LIN {X 0,Y 740.172,Z 409.434,A -85,B 0,C 180,E1 27946.505,E2 27946.505} C_VEL
LIN {X 0,Y 736.938,Z 402.446,A -85,B 0,C 180,E1 27945.781,E2 27945.781} C_VEL
LIN {X 0,Y 735.986,Z 399.553,A -85,B 0,C 180,E1 27945.49,E2 27945.49} C_VEL
LIN {X 0,Y 735.996,Z 399.549,A -85,B 0,C 180,E1 27943.152,E2 27943.152} C_VEL
LIN {X 0,Y 736.087,Z 399.542,A -85,B 0,C 180,E1 27940.285,E2 27940.285} C_VEL
LIN {X 0,Y 736.005,Z 399.54,A -85,B 0,C 180,E1 27937.589,E2 27937.589} C_VEL
LIN {X 0,Y 736,Z 399.544,A -85,B 0,C 180,E1 27935.266,E2 27935.266} C_VEL
LIN {X 0,Y 736.007,Z 399.541,A -85,B 0,C 180,E1 27933.009,E2 27933.009} C_VEL
LIN {X 0,Y 736.096,Z 399.538,A -85,B 0,C 180,E1 27930.24,E2 27930.24} C_VEL
LIN {X 0,Y 736.029,Z 399.541,A -85,B 0,C 180,E1 27927.421,E2 27927.421} C_VEL
LIN {X 0,Y 736.015,Z 399.535,A -85,B 0,C 180,E1 27924.993,E2 27924.993} C_VEL
LIN {X 0,Y 736.039,Z 399.543,A -85,B 0,C 180,E1 27922.518,E2 27922.518} C_VEL
LIN {X 0,Y 736.074,Z 399.535,A -85,B 0,C 180,E1 27919.485,E2 27919.485} C_VEL
LIN {X 0,Y 736.029,Z 399.54,A -85,B 0,C 180,E1 27916.82,E2 27916.82} C_VEL
LIN {X 0,Y 736.059,Z 399.536,A -85,B 0,C 180,E1 27914.234,E2 27914.234} C_VEL
LIN {X 0,Y 736.066,Z 399.535,A -85,B 0,C 180,E1 27911.122,E2 27911.122} C_VEL
LIN {X 0,Y 736.042,Z 399.533,A -85,B 0,C 180,E1 27908.437,E2 27908.437} C_VEL
LIN {X 0,Y 736.098,Z 399.541,A -85,B 0,C 180,E1 27905.691,E2 27905.691} C_VEL
LIN {X 0,Y 736.059,Z 399.529,A -85,B 0,C 180,E1 27902.725,E2 27902.725} C_VEL
LIN {X 0,Y 736.072,Z 399.542,A -85,B 0,C 180,E1 27899.922,E2 27899.922} C_VEL
LIN {X 0,Y 736.095,Z 399.525,A -85,B 0,C 180,E1 27896.885,E2 27896.885} C_VEL
LIN {X 0,Y 736.064,Z 399.54,A -85,B 0,C 180,E1 27893.996,E2 27893.996} C_VEL
LIN {X 0,Y 736.084,Z 399.532,A -85,B 0,C 180,E1 27891.17,E2 27891.17} C_VEL
LIN {X 0,Y 736.082,Z 399.538,A -85,B 0,C 180,E1 27889.085,E2 27889.085} C_VEL
LIN {X 0,Y 735.104,Z 399.658,A -85,B 0,C 180,E1 27888.486,E2 27888.486} C_VEL
LIN {X 0,Y 728.704,Z 400.452,A -85,B 0,C 180,E1 27886.806,E2 27886.806} C_VEL
LIN {X 0,Y 728.145,Z 400.519,A -85,B 0,C 180,E1 27886.37,E2 27886.37} C_VEL
LIN {X 0,Y 728.158,Z 400.528,A -85,B 0,C 180,E1 27883.404,E2 27883.404} C_VEL
LIN {X 0,Y 728.158,Z 400.516,A -85,B 0,C 180,E1 27880.34,E2 27880.34} C_VEL
LIN {X 0,Y 728.159,Z 400.532,A -85,B 0,C 180,E1 27877.303,E2 27877.303} C_VEL
LIN {X 0,Y 728.149,Z 400.514,A -85,B 0,C 180,E1 27874.265,E2 27874.265} C_VEL
LIN {X 0,Y 728.155,Z 400.529,A -85,B 0,C 180,E1 27871.174,E2 27871.174} C_VEL
LIN {X 0,Y 728.136,Z 400.524,A -85,B 0,C 180,E1 27868.214,E2 27868.214} C_VEL
LIN {X 0,Y 728.153,Z 400.524,A -85,B 0,C 180,E1 27865.202,E2 27865.202} C_VEL
LIN {X 0,Y 728.116,Z 400.521,A -85,B 0,C 180,E1 27862.331,E2 27862.331} C_VEL
LIN {X 0,Y 728.157,Z 400.526,A -85,B 0,C 180,E1 27859.495,E2 27859.495} C_VEL
LIN {X 0,Y 728.12,Z 400.535,A -85,B 0,C 180,E1 27856.528,E2 27856.528} C_VEL
LIN {X 0,Y 728.127,Z 400.666,A -85,B 0,C 180,E1 27854.303,E2 27854.303} C_VEL
LIN {X 0,Y 729.384,Z 403.968,A -85,B 0,C 180,E1 27853.969,E2 27853.969} C_VEL
LIN {X 0,Y 733.459,Z 413.169,A -85,B 0,C 180,E1 27853.013,E2 27853.013} C_VEL
LIN {X 0,Y 733.539,Z 418.371,A -85,B 0,C 180,E1 27852.673,E2 27852.673} C_VEL
LIN {X 0,Y 735.86,Z 427.418,A -85,B 0,C 180,E1 27852.39,E2 27852.39} C_VEL
LIN {X 0,Y 734.932,Z 640.42,A -85,B 0,C 180,E1 27849.748,E2 27849.748} C_VEL
LIN {X 0,Y 734.045,Z 865.401,A -85,B 0,C 180,E1 27847.051,E2 27847.051} C_VEL
LIN {X 0,Y 733.84,Z 901.954,A -85,B 0,C 180,E1 27846.581,E2 27846.581} C_VEL
LIN {X 0,Y 733.507,Z 929.139,A -85,B 0,C 180,E1 27846.067,E2 27846.067} C_VEL
LIN {X 0,Y 733.146,Z 955.092,A -85,B 0,C 180,E1 27845.422,E2 27845.422} C_VEL
LIN {X 0,Y 732.693,Z 983.223,A -85,B 0,C 180,E1 27844.544,E2 27844.544} C_VEL
LIN {X 0,Y 732.219,Z 1006.493,A -85,B 0,C 180,E1 27843.671,E2 27843.671} C_VEL
LIN {X 0,Y 731.801,Z 1027.689,A -85,B 0,C 180,E1 27842.757,E2 27842.757} C_VEL
LIN {X 0,Y 731.382,Z 1048.987,A -85,B 0,C 180,E1 27841.718,E2 27841.718} C_VEL
LIN {X 0,Y 730.847,Z 1074.292,A -85,B 0,C 180,E1 27840.312,E2 27840.312} C_VEL
LIN {X 0,Y 730.375,Z 1094.539,A -85,B 0,C 180,E1 27839.034,E2 27839.034} C_VEL
LIN {X 0,Y 730.006,Z 1112.829,A -85,B 0,C 180,E1 27837.757,E2 27837.757} C_VEL
LIN {X 0,Y 729.606,Z 1134.181,A -85,B 0,C 180,E1 27836.1,E2 27836.1} C_VEL
LIN {X 0,Y 729.201,Z 1151.944,A -85,B 0,C 180,E1 27834.551,E2 27834.551} C_VEL
LIN {X 0,Y 728.96,Z 1167.07,A -85,B 0,C 180,E1 27833.099,E2 27833.099} C_VEL
LIN {X 0,Y 728.696,Z 1184.595,A -85,B 0,C 180,E1 27831.24,E2 27831.24} C_VEL
LIN {X 0,Y 728.444,Z 1199.796,A -85,B 0,C 180,E1 27829.402,E2 27829.402} C_VEL
LIN {X 0,Y 728.27,Z 1211.506,A -85,B 0,C 180,E1 27827.83,E2 27827.83} C_VEL
LIN {X 0,Y 728.154,Z 1221.964,A -85,B 0,C 180,E1 27826.269,E2 27826.269} C_VEL
LIN {X 0,Y 728.097,Z 1232.189,A -85,B 0,C 180,E1 27824.557,E2 27824.557} C_VEL
LIN {X 0,Y 728.012,Z 1243.15,A -85,B 0,C 180,E1 27822.438,E2 27822.438} C_VEL
LIN {X 0,Y 727.956,Z 1251.705,A -85,B 0,C 180,E1 27820.431,E2 27820.431} C_VEL
LIN {X 0,Y 727.918,Z 1257.897,A -85,B 0,C 180,E1 27818.692,E2 27818.692} C_VEL
LIN {X 0,Y 727.914,Z 1263.45,A -85,B 0,C 180,E1 27816.786,E2 27816.786} C_VEL
LIN {X 0,Y 727.906,Z 1267.979,A -85,B 0,C 180,E1 27814.651,E2 27814.651} C_VEL
LIN {X 0,Y 727.907,Z 1270.635,A -85,B 0,C 180,E1 27812.6,E2 27812.6} C_VEL
LIN {X 0,Y 727.87,Z 1271.746,A -85,B 0,C 180,E1 27810.868,E2 27810.868} C_VEL
LIN {X 0,Y 727.863,Z 1271.818,A -85,B 0,C 180,E1 27809.294,E2 27809.294} C_VEL
LIN {X 0,Y 727.903,Z 1270.919,A -85,B 0,C 180,E1 27807.641,E2 27807.641} C_VEL
LIN {X 0,Y 727.919,Z 1268.753,A -85,B 0,C 180,E1 27805.749,E2 27805.749} C_VEL
LIN {X 0,Y 727.925,Z 1264.66,A -85,B 0,C 180,E1 27803.614,E2 27803.614} C_VEL
LIN {X 0,Y 727.938,Z 1258.97,A -85,B 0,C 180,E1 27801.551,E2 27801.551} C_VEL
LIN {X 0,Y 727.959,Z 1252.922,A -85,B 0,C 180,E1 27799.797,E2 27799.797} C_VEL
LIN {X 0,Y 727.968,Z 1246,A -85,B 0,C 180,E1 27798.113,E2 27798.113} C_VEL
LIN {X 0,Y 727.993,Z 1238.385,A -85,B 0,C 180,E1 27796.516,E2 27796.516} C_VEL
LIN {X 0,Y 728.083,Z 1229.937,A -85,B 0,C 180,E1 27794.959,E2 27794.959} C_VEL
LIN {X 0,Y 728.214,Z 1219.431,A -85,B 0,C 180,E1 27793.244,E2 27793.244} C_VEL
LIN {X 0,Y 728.406,Z 1204.399,A -85,B 0,C 180,E1 27791.101,E2 27791.101} C_VEL
LIN {X 0,Y 728.578,Z 1190.37,A -85,B 0,C 180,E1 27789.351,E2 27789.351} C_VEL
LIN {X 0,Y 728.782,Z 1176.161,A -85,B 0,C 180,E1 27787.752,E2 27787.752} C_VEL
LIN {X 0,Y 729.149,Z 1157.625,A -85,B 0,C 180,E1 27785.884,E2 27785.884} C_VEL
LIN {X 0,Y 729.437,Z 1139.857,A -85,B 0,C 180,E1 27784.292,E2 27784.292} C_VEL
LIN {X 0,Y 729.828,Z 1122.232,A -85,B 0,C 180,E1 27782.86,E2 27782.86} C_VEL
LIN {X 0,Y 730.303,Z 1099.259,A -85,B 0,C 180,E1 27781.192,E2 27781.192} C_VEL
LIN {X 0,Y 730.687,Z 1080.033,A -85,B 0,C 180,E1 27779.948,E2 27779.948} C_VEL
LIN {X 0,Y 731.122,Z 1060.07,A -85,B 0,C 180,E1 27778.784,E2 27778.784} C_VEL
LIN {X 0,Y 731.711,Z 1035.688,A -85,B 0,C 180,E1 27777.522,E2 27777.522} C_VEL
LIN {X 0,Y 732.155,Z 1010.998,A -85,B 0,C 180,E1 27776.425,E2 27776.425} C_VEL
LIN {X 0,Y 732.522,Z 990.893,A -85,B 0,C 180,E1 27775.642,E2 27775.642} C_VEL
LIN {X 0,Y 732.878,Z 969.752,A -85,B 0,C 180,E1 27774.927,E2 27774.927} C_VEL
LIN {X 0,Y 733.272,Z 946.183,A -85,B 0,C 180,E1 27774.25,E2 27774.25} C_VEL
LIN {X 0,Y 733.633,Z 919.552,A -85,B 0,C 180,E1 27773.644,E2 27773.644} C_VEL
LIN {X 0,Y 733.894,Z 892.765,A -85,B 0,C 180,E1 27773.194,E2 27773.194} C_VEL
LIN {X 0,Y 734.857,Z 657.43,A -85,B 0,C 180,E1 27770.369,E2 27770.369} C_VEL
LIN {X 0,Y 735.717,Z 452.431,A -85,B 0,C 180,E1 27767.834,E2 27767.834} C_VEL
LIN {X 0,Y 735.682,Z 426.075,A -85,B 0,C 180,E1 27767.49,E2 27767.49} C_VEL
LIN {X 0,Y 733.393,Z 417.703,A -85,B 0,C 180,E1 27767.209,E2 27767.209} C_VEL
LIN {X 0,Y 733.27,Z 412.662,A -85,B 0,C 180,E1 27766.847,E2 27766.847} C_VEL
LIN {X 0,Y 728.891,Z 403.155,A -85,B 0,C 180,E1 27765.845,E2 27765.845} C_VEL
LIN {X 0,Y 728.094,Z 400.538,A -85,B 0,C 180,E1 27765.571,E2 27765.571} C_VEL
LIN {X 0,Y 728.16,Z 400.529,A -85,B 0,C 180,E1 27762.715,E2 27762.715} C_VEL
LIN {X 0,Y 728.101,Z 400.53,A -85,B 0,C 180,E1 27759.862,E2 27759.862} C_VEL
LIN {X 0,Y 728.09,Z 400.531,A -85,B 0,C 180,E1 27757.339,E2 27757.339} C_VEL
LIN {X 0,Y 728.157,Z 400.524,A -85,B 0,C 180,E1 27754.53,E2 27754.53} C_VEL
LIN {X 0,Y 728.104,Z 400.526,A -85,B 0,C 180,E1 27751.641,E2 27751.641} C_VEL
LIN {X 0,Y 728.085,Z 400.526,A -85,B 0,C 180,E1 27749.088,E2 27749.088} C_VEL
LIN {X 0,Y 728.133,Z 400.532,A -85,B 0,C 180,E1 27746.419,E2 27746.419} C_VEL
LIN {X 0,Y 728.103,Z 400.528,A -85,B 0,C 180,E1 27743.383,E2 27743.383} C_VEL
LIN {X 0,Y 728.081,Z 400.525,A -85,B 0,C 180,E1 27740.92,E2 27740.92} C_VEL
LIN {X 0,Y 728.097,Z 400.529,A -85,B 0,C 180,E1 27738.403,E2 27738.403} C_VEL
LIN {X 0,Y 728.145,Z 400.517,A -85,B 0,C 180,E1 27735.442,E2 27735.442} C_VEL
LIN {X 0,Y 728.081,Z 400.528,A -85,B 0,C 180,E1 27732.774,E2 27732.774} C_VEL
LIN {X 0,Y 728.078,Z 400.529,A -85,B 0,C 180,E1 27730.364,E2 27730.364} C_VEL
LIN {X 0,Y 728.14,Z 400.525,A -85,B 0,C 180,E1 27727.655,E2 27727.655} C_VEL
LIN {X 0,Y 728.096,Z 400.526,A -85,B 0,C 180,E1 27724.726,E2 27724.726} C_VEL
LIN {X 0,Y 728.073,Z 400.522,A -85,B 0,C 180,E1 27722.283,E2 27722.283} C_VEL
LIN {X 0,Y 728.082,Z 400.532,A -85,B 0,C 180,E1 27719.843,E2 27719.843} C_VEL
LIN {X 0,Y 728.159,Z 400.52,A -85,B 0,C 180,E1 27716.93,E2 27716.93} C_VEL
LIN {X 0,Y 728.077,Z 400.53,A -85,B 0,C 180,E1 27714.167,E2 27714.167} C_VEL
LIN {X 0,Y 728.069,Z 400.528,A -85,B 0,C 180,E1 27711.788,E2 27711.788} C_VEL
LIN {X 0,Y 728.09,Z 400.527,A -85,B 0,C 180,E1 27709.316,E2 27709.316} C_VEL
LIN {X 0,Y 728.11,Z 400.524,A -85,B 0,C 180,E1 27706.256,E2 27706.256} C_VEL
LIN {X 0,Y 728.068,Z 400.527,A -85,B 0,C 180,E1 27703.716,E2 27703.716} C_VEL
LIN {X 0,Y 728.065,Z 400.531,A -85,B 0,C 180,E1 27701.357,E2 27701.357} C_VEL
LIN {X 0,Y 728.097,Z 400.524,A -85,B 0,C 180,E1 27698.827,E2 27698.827} C_VEL
LIN {X 0,Y 728.088,Z 400.527,A -85,B 0,C 180,E1 27695.754,E2 27695.754} C_VEL
LIN {X 0,Y 728.061,Z 400.53,A -85,B 0,C 180,E1 27693.315,E2 27693.315} C_VEL
LIN {X 0,Y 728.059,Z 400.531,A -85,B 0,C 180,E1 27691.091,E2 27691.091} C_VEL
LIN {X 0,Y 728.063,Z 400.53,A -85,B 0,C 180,E1 27688.817,E2 27688.817} C_VEL
LIN {X 0,Y 728.149,Z 400.526,A -85,B 0,C 180,E1 27686.03,E2 27686.03} C_VEL
LIN {X 0,Y 728.07,Z 400.533,A -85,B 0,C 180,E1 27683.186,E2 27683.186} C_VEL
LIN {X 0,Y 728.055,Z 400.535,A -85,B 0,C 180,E1 27680.82,E2 27680.82} C_VEL
LIN {X 0,Y 728.054,Z 400.529,A -85,B 0,C 180,E1 27678.55,E2 27678.55} C_VEL
LIN {X 0,Y 728.081,Z 400.539,A -85,B 0,C 180,E1 27676.09,E2 27676.09} C_VEL
LIN {X 0,Y 728.109,Z 400.757,A -85,B 0,C 180,E1 27675.02,E2 27675.02} C_VEL
LIN {X 0,Y 729.543,Z 404.285,A -85,B 0,C 180,E1 27674.657,E2 27674.657} C_VEL
LIN {X 0,Y 733.638,Z 413.428,A -85,B 0,C 180,E1 27673.704,E2 27673.704} C_VEL
LIN {X 0,Y 733.606,Z 428.254,A -85,B 0,C 180,E1 27672.715,E2 27672.715} C_VEL
LIN {X 0,Y 735.808,Z 437.166,A -85,B 0,C 180,E1 27672.442,E2 27672.442} C_VEL
LIN {X 0,Y 734.994,Z 637.58,A -85,B 0,C 180,E1 27669.949,E2 27669.949} C_VEL
LIN {X 0,Y 734.094,Z 863.168,A -85,B 0,C 180,E1 27667.24,E2 27667.24} C_VEL
LIN {X 0,Y 733.848,Z 909.112,A -85,B 0,C 180,E1 27666.669,E2 27666.669} C_VEL
LIN {X 0,Y 733.533,Z 936.271,A -85,B 0,C 180,E1 27666.174,E2 27666.174} C_VEL
LIN {X 0,Y 733.191,Z 962.414,A -85,B 0,C 180,E1 27665.54,E2 27665.54} C_VEL
LIN {X 0,Y 732.806,Z 987.825,A -85,B 0,C 180,E1 27664.77,E2 27664.77} C_VEL
LIN {X 0,Y 732.285,Z 1014.336,A -85,B 0,C 180,E1 27663.804,E2 27663.804} C_VEL
LIN {X 0,Y 731.832,Z 1035.781,A -85,B 0,C 180,E1 27662.89,E2 27662.89} C_VEL
LIN {X 0,Y 731.418,Z 1056.259,A -85,B 0,C 180,E1 27661.903,E2 27661.903} C_VEL
LIN {X 0,Y 730.988,Z 1078.915,A -85,B 0,C 180,E1 27660.674,E2 27660.674} C_VEL
LIN {X 0,Y 730.433,Z 1102.632,A -85,B 0,C 180,E1 27659.206,E2 27659.206} C_VEL
LIN {X 0,Y 730.019,Z 1121.699,A -85,B 0,C 180,E1 27657.884,E2 27657.884} C_VEL
LIN {X 0,Y 729.65,Z 1141.909,A -85,B 0,C 180,E1 27656.334,E2 27656.334} C_VEL
LIN {X 0,Y 729.212,Z 1161.552,A -85,B 0,C 180,E1 27654.632,E2 27654.632} C_VEL
LIN {X 0,Y 728.956,Z 1177.569,A -85,B 0,C 180,E1 27653.094,E2 27653.094} C_VEL
LIN {X 0,Y 728.684,Z 1195.015,A -85,B 0,C 180,E1 27651.235,E2 27651.235} C_VEL
LIN {X 0,Y 728.438,Z 1210.181,A -85,B 0,C 180,E1 27649.398,E2 27649.398} C_VEL
LIN {X 0,Y 728.264,Z 1221.856,A -85,B 0,C 180,E1 27647.826,E2 27647.826} C_VEL
LIN {X 0,Y 728.149,Z 1232.802,A -85,B 0,C 180,E1 27646.183,E2 27646.183} C_VEL
LIN {X 0,Y 728.085,Z 1244.324,A -85,B 0,C 180,E1 27644.227,E2 27644.227} C_VEL
LIN {X 0,Y 727.973,Z 1254.727,A -85,B 0,C 180,E1 27642.128,E2 27642.128} C_VEL
LIN {X 0,Y 727.956,Z 1261.878,A -85,B 0,C 180,E1 27640.431,E2 27640.431} C_VEL
LIN {X 0,Y 727.915,Z 1267.801,A -85,B 0,C 180,E1 27638.768,E2 27638.768} C_VEL
LIN {X 0,Y 727.918,Z 1273.181,A -85,B 0,C 180,E1 27636.94,E2 27636.94} C_VEL
LIN {X 0,Y 727.911,Z 1277.787,A -85,B 0,C 180,E1 27634.804,E2 27634.804} C_VEL
LIN {X 0,Y 727.913,Z 1280.543,A -85,B 0,C 180,E1 27632.753,E2 27632.753} C_VEL
LIN {X 0,Y 727.874,Z 1281.715,A -85,B 0,C 180,E1 27631.021,E2 27631.021} C_VEL
LIN {X 0,Y 727.863,Z 1281.826,A -85,B 0,C 180,E1 27629.368,E2 27629.368} C_VEL
LIN {X 0,Y 727.907,Z 1280.944,A -85,B 0,C 180,E1 27627.715,E2 27627.715} C_VEL
LIN {X 0,Y 727.919,Z 1278.799,A -85,B 0,C 180,E1 27625.823,E2 27625.823} C_VEL
LIN {X 0,Y 727.925,Z 1274.73,A -85,B 0,C 180,E1 27623.689,E2 27623.689} C_VEL
LIN {X 0,Y 727.94,Z 1269.067,A -85,B 0,C 180,E1 27621.626,E2 27621.626} C_VEL
LIN {X 0,Y 727.957,Z 1263.038,A -85,B 0,C 180,E1 27619.872,E2 27619.872} C_VEL
LIN {X 0,Y 727.966,Z 1256.136,A -85,B 0,C 180,E1 27618.189,E2 27618.189} C_VEL
LIN {X 0,Y 727.992,Z 1248.874,A -85,B 0,C 180,E1 27616.657,E2 27616.657} C_VEL
LIN {X 0,Y 728.086,Z 1240.585,A -85,B 0,C 180,E1 27615.118,E2 27615.118} C_VEL
LIN {X 0,Y 728.176,Z 1230.683,A -85,B 0,C 180,E1 27613.485,E2 27613.485} C_VEL
LIN {X 0,Y 728.348,Z 1218.33,A -85,B 0,C 180,E1 27611.675,E2 27611.675} C_VEL
LIN {X 0,Y 728.544,Z 1202.255,A -85,B 0,C 180,E1 27609.617,E2 27609.617} C_VEL
LIN {X 0,Y 728.751,Z 1188.504,A -85,B 0,C 180,E1 27608.051,E2 27608.051} C_VEL
LIN {X 0,Y 729.019,Z 1173.252,A -85,B 0,C 180,E1 27606.475,E2 27606.475} C_VEL
LIN {X 0,Y 729.419,Z 1152.829,A -85,B 0,C 180,E1 27604.591,E2 27604.591} C_VEL
LIN {X 0,Y 729.707,Z 1136.033,A -85,B 0,C 180,E1 27603.203,E2 27603.203} C_VEL
LIN {X 0,Y 730.116,Z 1118.042,A -85,B 0,C 180,E1 27601.851,E2 27601.851} C_VEL
LIN {X 0,Y 730.637,Z 1095.045,A -85,B 0,C 180,E1 27600.303,E2 27600.303} C_VEL
LIN {X 0,Y 731.035,Z 1073.976,A -85,B 0,C 180,E1 27599.048,E2 27599.048} C_VEL
LIN {X 0,Y 731.459,Z 1053.715,A -85,B 0,C 180,E1 27597.967,E2 27597.967} C_VEL
LIN {X 0,Y 732.011,Z 1030.233,A -85,B 0,C 180,E1 27596.859,E2 27596.859} C_VEL
LIN {X 0,Y 732.493,Z 1004.359,A -85,B 0,C 180,E1 27595.815,E2 27595.815} C_VEL
LIN {X 0,Y 732.86,Z 982.526,A -85,B 0,C 180,E1 27595.061,E2 27595.061} C_VEL
LIN {X 0,Y 733.226,Z 959.937,A -85,B 0,C 180,E1 27594.393,E2 27594.393} C_VEL
LIN {X 0,Y 733.593,Z 933.231,A -85,B 0,C 180,E1 27593.762,E2 27593.762} C_VEL
LIN {X 0,Y 733.868,Z 905.776,A -85,B 0,C 180,E1 27593.281,E2 27593.281} C_VEL
LIN {X 0,Y 734.847,Z 670.065,A -85,B 0,C 180,E1 27590.446,E2 27590.446} C_VEL
LIN {X 0,Y 735.657,Z 471.261,A -85,B 0,C 180,E1 27587.988,E2 27587.988} C_VEL
LIN {X 0,Y 735.65,Z 435.773,A -85,B 0,C 180,E1 27587.529,E2 27587.529} C_VEL
LIN {X 0,Y 733.473,Z 427.342,A -85,B 0,C 180,E1 27587.243,E2 27587.243} C_VEL
LIN {X 0,Y 733.521,Z 413.008,A -85,B 0,C 180,E1 27586.259,E2 27586.259} C_VEL
LIN {X 0,Y 728.16,Z 401.076,A -85,B 0,C 180,E1 27585.007,E2 27585.007} C_VEL
LIN {X 0,Y 728.082,Z 400.54,A -85,B 0,C 180,E1 27584.938,E2 27584.938} C_VEL
LIN {X 0,Y 728.072,Z 400.531,A -85,B 0,C 180,E1 27581.87,E2 27581.87} C_VEL
LIN {X 0,Y 728.055,Z 400.536,A -85,B 0,C 180,E1 27579.481,E2 27579.481} C_VEL
LIN {X 0,Y 728.06,Z 400.529,A -85,B 0,C 180,E1 27577.177,E2 27577.177} C_VEL
LIN {X 0,Y 728.102,Z 400.534,A -85,B 0,C 180,E1 27574.649,E2 27574.649} C_VEL
LIN {X 0,Y 728.094,Z 400.53,A -85,B 0,C 180,E1 27571.631,E2 27571.631} C_VEL
LIN {X 0,Y 728.071,Z 400.527,A -85,B 0,C 180,E1 27569.139,E2 27569.139} C_VEL
LIN {X 0,Y 728.083,Z 400.532,A -85,B 0,C 180,E1 27566.773,E2 27566.773} C_VEL
LIN {X 0,Y 728.161,Z 400.528,A -85,B 0,C 180,E1 27563.861,E2 27563.861} C_VEL
LIN {X 0,Y 728.09,Z 400.525,A -85,B 0,C 180,E1 27561.088,E2 27561.088} C_VEL
LIN {X 0,Y 728.095,Z 400.528,A -85,B 0,C 180,E1 27558.579,E2 27558.579} C_VEL
LIN {X 0,Y 728.159,Z 400.518,A -85,B 0,C 180,E1 27555.695,E2 27555.695} C_VEL
LIN {X 0,Y 728.1,Z 400.527,A -85,B 0,C 180,E1 27552.832,E2 27552.832} C_VEL
LIN {X 0,Y 728.127,Z 400.531,A -85,B 0,C 180,E1 27550.124,E2 27550.124} C_VEL
LIN {X 0,Y 728.133,Z 400.523,A -85,B 0,C 180,E1 27547.02,E2 27547.02} C_VEL
LIN {X 0,Y 728.113,Z 400.528,A -85,B 0,C 180,E1 27544.253,E2 27544.253} C_VEL
LIN {X 0,Y 728.152,Z 400.528,A -85,B 0,C 180,E1 27541.416,E2 27541.416} C_VEL
LIN {X 0,Y 728.124,Z 400.523,A -85,B 0,C 180,E1 27538.584,E2 27538.584} C_VEL
LIN {X 0,Y 728.145,Z 400.524,A -85,B 0,C 180,E1 27535.747,E2 27535.747} C_VEL
LIN {X 0,Y 728.153,Z 400.519,A -85,B 0,C 180,E1 27532.663,E2 27532.663} C_VEL
LIN {X 0,Y 728.147,Z 400.524,A -85,B 0,C 180,E1 27529.637,E2 27529.637} C_VEL
LIN {X 0,Y 728.159,Z 400.518,A -85,B 0,C 180,E1 27526.581,E2 27526.581} C_VEL
LIN {X 0,Y 728.145,Z 400.519,A -85,B 0,C 180,E1 27526.37,E2 27526.37} C_VEL
LIN {X 0,Y 727.117,Z 400.655,A -85,B 0,C 180,E1 27525.764,E2 27525.764} C_VEL
LIN {X 0,Y 720.707,Z 401.444,A -85,B 0,C 180,E1 27524.066,E2 27524.066} C_VEL
LIN {X 0,Y 720.204,Z 401.513,A -85,B 0,C 180,E1 27523.625,E2 27523.625} C_VEL
LIN {X 0,Y 720.2,Z 401.508,A -85,B 0,C 180,E1 27520.705,E2 27520.705} C_VEL
LIN {X 0,Y 720.199,Z 401.513,A -85,B 0,C 180,E1 27517.813,E2 27517.813} C_VEL
LIN {X 0,Y 720.198,Z 401.509,A -85,B 0,C 180,E1 27514.947,E2 27514.947} C_VEL
LIN {X 0,Y 720.22,Z 401.511,A -85,B 0,C 180,E1 27512.002,E2 27512.002} C_VEL
LIN {X 0,Y 720.204,Z 401.518,A -85,B 0,C 180,E1 27508.938,E2 27508.938} C_VEL
LIN {X 0,Y 720.21,Z 401.505,A -85,B 0,C 180,E1 27505.979,E2 27505.979} C_VEL
LIN {X 0,Y 720.201,Z 401.514,A -85,B 0,C 180,E1 27502.836,E2 27502.836} C_VEL
LIN {X 0,Y 720.196,Z 401.515,A -85,B 0,C 180,E1 27499.906,E2 27499.906} C_VEL
LIN {X 0,Y 720.206,Z 401.523,A -85,B 0,C 180,E1 27496.793,E2 27496.793} C_VEL
LIN {X 0,Y 720.228,Z 401.618,A -85,B 0,C 180,E1 27494.851,E2 27494.851} C_VEL
LIN {X 0,Y 721.644,Z 405.235,A -85,B 0,C 180,E1 27494.474,E2 27494.474} C_VEL
LIN {X 0,Y 726.876,Z 417.505,A -85,B 0,C 180,E1 27493.191,E2 27493.191} C_VEL
LIN {X 0,Y 729.928,Z 429.522,A -85,B 0,C 180,E1 27492.789,E2 27492.789} C_VEL
LIN {X 0,Y 728.768,Z 641.616,A -85,B 0,C 180,E1 27490.138,E2 27490.138} C_VEL
LIN {X 0,Y 727.652,Z 866.412,A -85,B 0,C 180,E1 27487.42,E2 27487.42} C_VEL
LIN {X 0,Y 727.395,Z 902.179,A -85,B 0,C 180,E1 27486.955,E2 27486.955} C_VEL
LIN {X 0,Y 726.977,Z 929.413,A -85,B 0,C 180,E1 27486.436,E2 27486.436} C_VEL
LIN {X 0,Y 726.54,Z 955.115,A -85,B 0,C 180,E1 27485.794,E2 27485.794} C_VEL
LIN {X 0,Y 725.973,Z 983.236,A -85,B 0,C 180,E1 27484.91,E2 27484.91} C_VEL
LIN {X 0,Y 725.391,Z 1006.511,A -85,B 0,C 180,E1 27484.032,E2 27484.032} C_VEL
LIN {X 0,Y 724.843,Z 1027.705,A -85,B 0,C 180,E1 27483.112,E2 27483.112} C_VEL
LIN {X 0,Y 724.296,Z 1049.98,A -85,B 0,C 180,E1 27482.014,E2 27482.014} C_VEL
LIN {X 0,Y 723.62,Z 1075.255,A -85,B 0,C 180,E1 27480.587,E2 27480.587} C_VEL
LIN {X 0,Y 723.048,Z 1095.212,A -85,B 0,C 180,E1 27479.311,E2 27479.311} C_VEL
LIN {X 0,Y 722.555,Z 1114.047,A -85,B 0,C 180,E1 27477.978,E2 27477.978} C_VEL
LIN {X 0,Y 721.99,Z 1136.686,A -85,B 0,C 180,E1 27476.178,E2 27476.178} C_VEL
LIN {X 0,Y 721.541,Z 1153.317,A -85,B 0,C 180,E1 27474.701,E2 27474.701} C_VEL
LIN {X 0,Y 721.205,Z 1170.48,A -85,B 0,C 180,E1 27473.016,E2 27473.016} C_VEL
LIN {X 0,Y 720.826,Z 1188.154,A -85,B 0,C 180,E1 27471.057,E2 27471.057} C_VEL
LIN {X 0,Y 720.575,Z 1201.092,A -85,B 0,C 180,E1 27469.454,E2 27469.454} C_VEL
LIN {X 0,Y 720.364,Z 1212.676,A -85,B 0,C 180,E1 27467.865,E2 27467.865} C_VEL
LIN {X 0,Y 720.209,Z 1224.581,A -85,B 0,C 180,E1 27466.04,E2 27466.04} C_VEL
LIN {X 0,Y 720.07,Z 1236.598,A -85,B 0,C 180,E1 27463.902,E2 27463.902} C_VEL
LIN {X 0,Y 719.991,Z 1245.225,A -85,B 0,C 180,E1 27462.107,E2 27462.107} C_VEL
LIN {X 0,Y 719.969,Z 1252.256,A -85,B 0,C 180,E1 27460.403,E2 27460.403} C_VEL
LIN {X 0,Y 719.922,Z 1258.155,A -85,B 0,C 180,E1 27458.709,E2 27458.709} C_VEL
LIN {X 0,Y 719.917,Z 1263.646,A -85,B 0,C 180,E1 27456.782,E2 27456.782} C_VEL
LIN {X 0,Y 719.908,Z 1267.98,A -85,B 0,C 180,E1 27454.702,E2 27454.702} C_VEL
LIN {X 0,Y 719.908,Z 1270.636,A -85,B 0,C 180,E1 27452.629,E2 27452.629} C_VEL
LIN {X 0,Y 719.871,Z 1271.746,A -85,B 0,C 180,E1 27450.878,E2 27450.878} C_VEL
LIN {X 0,Y 719.863,Z 1271.818,A -85,B 0,C 180,E1 27449.286,E2 27449.286} C_VEL
LIN {X 0,Y 719.903,Z 1270.919,A -85,B 0,C 180,E1 27447.614,E2 27447.614} C_VEL
LIN {X 0,Y 719.918,Z 1268.752,A -85,B 0,C 180,E1 27445.701,E2 27445.701} C_VEL
LIN {X 0,Y 719.926,Z 1264.659,A -85,B 0,C 180,E1 27443.543,E2 27443.543} C_VEL
LIN {X 0,Y 719.944,Z 1258.919,A -85,B 0,C 180,E1 27441.441,E2 27441.441} C_VEL
LIN {X 0,Y 719.97,Z 1252.921,A -85,B 0,C 180,E1 27439.682,E2 27439.682} C_VEL
LIN {X 0,Y 719.988,Z 1246.356,A -85,B 0,C 180,E1 27438.061,E2 27438.061} C_VEL
LIN {X 0,Y 720.024,Z 1239.125,A -85,B 0,C 180,E1 27436.512,E2 27436.512} C_VEL
LIN {X 0,Y 720.131,Z 1230.867,A -85,B 0,C 180,E1 27434.954,E2 27434.954} C_VEL
LIN {X 0,Y 720.269,Z 1220.997,A -85,B 0,C 180,E1 27433.303,E2 27433.303} C_VEL
LIN {X 0,Y 720.453,Z 1209.259,A -85,B 0,C 180,E1 27431.556,E2 27431.556} C_VEL
LIN {X 0,Y 720.717,Z 1193.21,A -85,B 0,C 180,E1 27429.455,E2 27429.455} C_VEL
LIN {X 0,Y 720.984,Z 1178.498,A -85,B 0,C 180,E1 27427.756,E2 27427.756} C_VEL
LIN {X 0,Y 721.333,Z 1163.489,A -85,B 0,C 180,E1 27426.188,E2 27426.188} C_VEL
LIN {X 0,Y 721.809,Z 1143.406,A -85,B 0,C 180,E1 27424.309,E2 27424.309} C_VEL
LIN {X 0,Y 722.247,Z 1125.548,A -85,B 0,C 180,E1 27422.82,E2 27422.82} C_VEL
LIN {X 0,Y 722.763,Z 1106.86,A -85,B 0,C 180,E1 27421.406,E2 27421.406} C_VEL
LIN {X 0,Y 723.392,Z 1082.938,A -85,B 0,C 180,E1 27419.797,E2 27419.797} C_VEL
LIN {X 0,Y 723.923,Z 1062.552,A -85,B 0,C 180,E1 27418.582,E2 27418.582} C_VEL
LIN {X 0,Y 724.507,Z 1041.94,A -85,B 0,C 180,E1 27417.484,E2 27417.484} C_VEL
LIN {X 0,Y 725.209,Z 1016.579,A -85,B 0,C 180,E1 27416.297,E2 27416.297} C_VEL
LIN {X 0,Y 725.728,Z 992.151,A -85,B 0,C 180,E1 27415.323,E2 27415.323} C_VEL
LIN {X 0,Y 726.176,Z 971.162,A -85,B 0,C 180,E1 27414.602,E2 27414.602} C_VEL
LIN {X 0,Y 726.658,Z 948.013,A -85,B 0,C 180,E1 27413.924,E2 27413.924} C_VEL
LIN {X 0,Y 727.128,Z 920.985,A -85,B 0,C 180,E1 27413.295,E2 27413.295} C_VEL
LIN {X 0,Y 727.456,Z 893.868,A -85,B 0,C 180,E1 27412.831,E2 27412.831} C_VEL
LIN {X 0,Y 728.662,Z 661.18,A -85,B 0,C 180,E1 27410.012,E2 27410.012} C_VEL
LIN {X 0,Y 729.743,Z 456.973,A -85,B 0,C 180,E1 27407.467,E2 27407.467} C_VEL
LIN {X 0,Y 729.758,Z 428.221,A -85,B 0,C 180,E1 27407.091,E2 27407.091} C_VEL
LIN {X 0,Y 726.861,Z 417.589,A -85,B 0,C 180,E1 27406.724,E2 27406.724} C_VEL
LIN {X 0,Y 725.811,Z 414.683,A -85,B 0,C 180,E1 27406.438,E2 27406.438} C_VEL
LIN {X 0,Y 720.341,Z 402.352,A -85,B 0,C 180,E1 27405.123,E2 27405.123} C_VEL
LIN {X 0,Y 720.206,Z 401.523,A -85,B 0,C 180,E1 27405.042,E2 27405.042} C_VEL
LIN {X 0,Y 720.169,Z 401.514,A -85,B 0,C 180,E1 27402.007,E2 27402.007} C_VEL
LIN {X 0,Y 720.151,Z 401.522,A -85,B 0,C 180,E1 27399.475,E2 27399.475} C_VEL
LIN {X 0,Y 720.202,Z 401.521,A -85,B 0,C 180,E1 27396.754,E2 27396.754} C_VEL
LIN {X 0,Y 720.167,Z 401.513,A -85,B 0,C 180,E1 27393.736,E2 27393.736} C_VEL
LIN {X 0,Y 720.147,Z 401.518,A -85,B 0,C 180,E1 27391.191,E2 27391.191} C_VEL
LIN {X 0,Y 720.189,Z 401.517,A -85,B 0,C 180,E1 27388.529,E2 27388.529} C_VEL
LIN {X 0,Y 720.168,Z 401.507,A -85,B 0,C 180,E1 27385.494,E2 27385.494} C_VEL
LIN {X 0,Y 720.143,Z 401.519,A -85,B 0,C 180,E1 27382.964,E2 27382.964} C_VEL
LIN {X 0,Y 720.167,Z 401.516,A -85,B 0,C 180,E1 27380.395,E2 27380.395} C_VEL
LIN {X 0,Y 720.175,Z 401.516,A -85,B 0,C 180,E1 27377.285,E2 27377.285} C_VEL
LIN {X 0,Y 720.138,Z 401.508,A -85,B 0,C 180,E1 27374.72,E2 27374.72} C_VEL
LIN {X 0,Y 720.149,Z 401.52,A -85,B 0,C 180,E1 27372.265,E2 27372.265} C_VEL
LIN {X 0,Y 720.219,Z 401.505,A -85,B 0,C 180,E1 27369.348,E2 27369.348} C_VEL
LIN {X 0,Y 720.14,Z 401.518,A -85,B 0,C 180,E1 27366.538,E2 27366.538} C_VEL
LIN {X 0,Y 720.137,Z 401.518,A -85,B 0,C 180,E1 27364.14,E2 27364.14} C_VEL
LIN {X 0,Y 720.2,Z 401.513,A -85,B 0,C 180,E1 27361.432,E2 27361.432} C_VEL
LIN {X 0,Y 720.152,Z 401.515,A -85,B 0,C 180,E1 27358.488,E2 27358.488} C_VEL
LIN {X 0,Y 720.13,Z 401.512,A -85,B 0,C 180,E1 27356.019,E2 27356.019} C_VEL
LIN {X 0,Y 720.139,Z 401.521,A -85,B 0,C 180,E1 27353.623,E2 27353.623} C_VEL
LIN {X 0,Y 720.219,Z 401.508,A -85,B 0,C 180,E1 27350.732,E2 27350.732} C_VEL
LIN {X 0,Y 720.133,Z 401.52,A -85,B 0,C 180,E1 27347.897,E2 27347.897} C_VEL
LIN {X 0,Y 720.127,Z 401.515,A -85,B 0,C 180,E1 27345.527,E2 27345.527} C_VEL
LIN {X 0,Y 720.153,Z 401.518,A -85,B 0,C 180,E1 27343.048,E2 27343.048} C_VEL
LIN {X 0,Y 720.155,Z 401.508,A -85,B 0,C 180,E1 27339.944,E2 27339.944} C_VEL
LIN {X 0,Y 720.126,Z 401.52,A -85,B 0,C 180,E1 27337.466,E2 27337.466} C_VEL
LIN {X 0,Y 720.124,Z 401.517,A -85,B 0,C 180,E1 27335.12,E2 27335.12} C_VEL
LIN {X 0,Y 720.168,Z 401.521,A -85,B 0,C 180,E1 27332.512,E2 27332.512} C_VEL
LIN {X 0,Y 720.148,Z 401.518,A -85,B 0,C 180,E1 27329.55,E2 27329.55} C_VEL
LIN {X 0,Y 720.121,Z 401.521,A -85,B 0,C 180,E1 27327.118,E2 27327.118} C_VEL
LIN {X 0,Y 720.118,Z 401.521,A -85,B 0,C 180,E1 27324.814,E2 27324.814} C_VEL
LIN {X 0,Y 720.141,Z 401.523,A -85,B 0,C 180,E1 27322.343,E2 27322.343} C_VEL
LIN {X 0,Y 720.152,Z 401.513,A -85,B 0,C 180,E1 27319.264,E2 27319.264} C_VEL
LIN {X 0,Y 720.119,Z 401.529,A -85,B 0,C 180,E1 27316.793,E2 27316.793} C_VEL
LIN {X 0,Y 720.215,Z 401.53,A -85,B 0,C 180,E1 27315.596,E2 27315.596} C_VEL
LIN {X 0,Y 721.448,Z 404.969,A -85,B 0,C 180,E1 27315.246,E2 27315.246} C_VEL
LIN {X 0,Y 727.108,Z 417.692,A -85,B 0,C 180,E1 27313.897,E2 27313.897} C_VEL
LIN {X 0,Y 727.068,Z 428.227,A -85,B 0,C 180,E1 27313.193,E2 27313.193} C_VEL
LIN {X 0,Y 729.88,Z 439.222,A -85,B 0,C 180,E1 27312.842,E2 27312.842} C_VEL
LIN {X 0,Y 728.84,Z 639.374,A -85,B 0,C 180,E1 27310.333,E2 27310.333} C_VEL
LIN {X 0,Y 727.709,Z 865.076,A -85,B 0,C 180,E1 27307.6,E2 27307.6} C_VEL
LIN {X 0,Y 727.404,Z 909.707,A -85,B 0,C 180,E1 27307.038,E2 27307.038} C_VEL
LIN {X 0,Y 727.015,Z 936.924,A -85,B 0,C 180,E1 27306.536,E2 27306.536} C_VEL
LIN {X 0,Y 726.583,Z 962.722,A -85,B 0,C 180,E1 27305.904,E2 27305.904} C_VEL
LIN {X 0,Y 726.094,Z 988.507,A -85,B 0,C 180,E1 27305.116,E2 27305.116} C_VEL
LIN {X 0,Y 725.429,Z 1015.457,A -85,B 0,C 180,E1 27304.119,E2 27304.119} C_VEL
LIN {X 0,Y 724.873,Z 1036.778,A -85,B 0,C 180,E1 27303.199,E2 27303.199} C_VEL
LIN {X 0,Y 724.34,Z 1057.382,A -85,B 0,C 180,E1 27302.193,E2 27302.193} C_VEL
LIN {X 0,Y 723.766,Z 1081.272,A -85,B 0,C 180,E1 27300.875,E2 27300.875} C_VEL
LIN {X 0,Y 723.115,Z 1103.296,A -85,B 0,C 180,E1 27299.485,E2 27299.485} C_VEL
LIN {X 0,Y 722.604,Z 1121.865,A -85,B 0,C 180,E1 27298.183,E2 27298.183} C_VEL
LIN {X 0,Y 722.104,Z 1142.726,A -85,B 0,C 180,E1 27296.564,E2 27296.564} C_VEL
LIN {X 0,Y 721.584,Z 1162.018,A -85,B 0,C 180,E1 27294.866,E2 27294.866} C_VEL
LIN {X 0,Y 721.236,Z 1177.57,A -85,B 0,C 180,E1 27293.356,E2 27293.356} C_VEL
LIN {X 0,Y 720.893,Z 1195.177,A -85,B 0,C 180,E1 27291.457,E2 27291.457} C_VEL
LIN {X 0,Y 720.586,Z 1210.183,A -85,B 0,C 180,E1 27289.618,E2 27289.618} C_VEL
LIN {X 0,Y 720.383,Z 1221.858,A -85,B 0,C 180,E1 27288.027,E2 27288.027} C_VEL
LIN {X 0,Y 720.226,Z 1232.804,A -85,B 0,C 180,E1 27286.366,E2 27286.366} C_VEL
LIN {X 0,Y 720.133,Z 1244.323,A -85,B 0,C 180,E1 27284.388,E2 27284.388} C_VEL
LIN {X 0,Y 720.005,Z 1254.729,A -85,B 0,C 180,E1 27282.264,E2 27282.264} C_VEL
LIN {X 0,Y 719.961,Z 1261.832,A -85,B 0,C 180,E1 27280.561,E2 27280.561} C_VEL
LIN {X 0,Y 719.912,Z 1267.801,A -85,B 0,C 180,E1 27278.866,E2 27278.866} C_VEL
LIN {X 0,Y 719.923,Z 1273.181,A -85,B 0,C 180,E1 27277.018,E2 27277.018} C_VEL
LIN {X 0,Y 719.914,Z 1277.787,A -85,B 0,C 180,E1 27274.858,E2 27274.858} C_VEL
LIN {X 0,Y 719.914,Z 1280.543,A -85,B 0,C 180,E1 27272.784,E2 27272.784} C_VEL
LIN {X 0,Y 719.875,Z 1281.715,A -85,B 0,C 180,E1 27271.032,E2 27271.032} C_VEL
LIN {X 0,Y 719.863,Z 1281.826,A -85,B 0,C 180,E1 27269.361,E2 27269.361} C_VEL
LIN {X 0,Y 719.906,Z 1280.944,A -85,B 0,C 180,E1 27267.689,E2 27267.689} C_VEL
LIN {X 0,Y 719.919,Z 1278.799,A -85,B 0,C 180,E1 27265.776,E2 27265.776} C_VEL
LIN {X 0,Y 719.926,Z 1274.73,A -85,B 0,C 180,E1 27263.619,E2 27263.619} C_VEL
LIN {X 0,Y 719.944,Z 1269.067,A -85,B 0,C 180,E1 27261.532,E2 27261.532} C_VEL
LIN {X 0,Y 719.969,Z 1263.038,A -85,B 0,C 180,E1 27259.759,E2 27259.759} C_VEL
LIN {X 0,Y 719.986,Z 1256.137,A -85,B 0,C 180,E1 27258.056,E2 27258.056} C_VEL
LIN {X 0,Y 720.023,Z 1248.875,A -85,B 0,C 180,E1 27256.507,E2 27256.507} C_VEL
LIN {X 0,Y 720.135,Z 1240.587,A -85,B 0,C 180,E1 27254.949,E2 27254.949} C_VEL
LIN {X 0,Y 720.273,Z 1230.685,A -85,B 0,C 180,E1 27253.299,E2 27253.299} C_VEL
LIN {X 0,Y 720.5,Z 1217.167,A -85,B 0,C 180,E1 27251.301,E2 27251.301} C_VEL
LIN {X 0,Y 720.738,Z 1202.082,A -85,B 0,C 180,E1 27249.366,E2 27249.366} C_VEL
LIN {X 0,Y 720.993,Z 1188.044,A -85,B 0,C 180,E1 27247.752,E2 27247.752} C_VEL
LIN {X 0,Y 721.368,Z 1172.4,A -85,B 0,C 180,E1 27246.124,E2 27246.124} C_VEL
LIN {X 0,Y 721.823,Z 1152.321,A -85,B 0,C 180,E1 27244.26,E2 27244.26} C_VEL
LIN {X 0,Y 722.271,Z 1134.926,A -85,B 0,C 180,E1 27242.815,E2 27242.815} C_VEL
LIN {X 0,Y 722.803,Z 1115.574,A -85,B 0,C 180,E1 27241.357,E2 27241.357} C_VEL
LIN {X 0,Y 723.401,Z 1092.137,A -85,B 0,C 180,E1 27239.792,E2 27239.792} C_VEL
LIN {X 0,Y 723.939,Z 1072.106,A -85,B 0,C 180,E1 27238.603,E2 27238.603} C_VEL
LIN {X 0,Y 724.543,Z 1050.966,A -85,B 0,C 180,E1 27237.48,E2 27237.48} C_VEL
LIN {X 0,Y 725.224,Z 1025.392,A -85,B 0,C 180,E1 27236.293,E2 27236.293} C_VEL
LIN {X 0,Y 725.73,Z 1002.083,A -85,B 0,C 180,E1 27235.365,E2 27235.365} C_VEL
LIN {X 0,Y 726.181,Z 981.062,A -85,B 0,C 180,E1 27234.644,E2 27234.644} C_VEL
LIN {X 0,Y 726.657,Z 958.072,A -85,B 0,C 180,E1 27233.97,E2 27233.97} C_VEL
LIN {X 0,Y 727.127,Z 931.124,A -85,B 0,C 180,E1 27233.343,E2 27233.343} C_VEL
LIN {X 0,Y 727.456,Z 903.893,A -85,B 0,C 180,E1 27232.876,E2 27232.876} C_VEL
LIN {X 0,Y 728.668,Z 670.32,A -85,B 0,C 180,E1 27230.047,E2 27230.047} C_VEL
LIN {X 0,Y 729.699,Z 471.578,A -85,B 0,C 180,E1 27227.569,E2 27227.569} C_VEL
LIN {X 0,Y 729.73,Z 437.882,A -85,B 0,C 180,E1 27227.13,E2 27227.13} C_VEL
LIN {X 0,Y 726.945,Z 427.342,A -85,B 0,C 180,E1 27226.765,E2 27226.765} C_VEL
LIN {X 0,Y 727.026,Z 417.068,A -85,B 0,C 180,E1 27226.053,E2 27226.053} C_VEL
LIN {X 0,Y 720.377,Z 402.446,A -85,B 0,C 180,E1 27224.484,E2 27224.484} C_VEL
LIN {X 0,Y 720.197,Z 401.524,A -85,B 0,C 180,E1 27224.378,E2 27224.378} C_VEL
LIN {X 0,Y 720.114,Z 401.52,A -85,B 0,C 180,E1 27221.584,E2 27221.584} C_VEL
LIN {X 0,Y 720.116,Z 401.526,A -85,B 0,C 180,E1 27219.284,E2 27219.284} C_VEL
LIN {X 0,Y 720.151,Z 401.518,A -85,B 0,C 180,E1 27216.757,E2 27216.757} C_VEL
LIN {X 0,Y 720.146,Z 401.517,A -85,B 0,C 180,E1 27213.642,E2 27213.642} C_VEL
LIN {X 0,Y 720.13,Z 401.52,A -85,B 0,C 180,E1 27211.192,E2 27211.192} C_VEL
LIN {X 0,Y 720.142,Z 401.517,A -85,B 0,C 180,E1 27208.803,E2 27208.803} C_VEL
LIN {X 0,Y 720.216,Z 401.507,A -85,B 0,C 180,E1 27205.891,E2 27205.891} C_VEL
LIN {X 0,Y 720.146,Z 401.519,A -85,B 0,C 180,E1 27203.137,E2 27203.137} C_VEL
LIN {X 0,Y 720.152,Z 401.515,A -85,B 0,C 180,E1 27200.641,E2 27200.641} C_VEL
LIN {X 0,Y 720.223,Z 401.517,A -85,B 0,C 180,E1 27197.755,E2 27197.755} C_VEL
LIN {X 0,Y 720.156,Z 401.506,A -85,B 0,C 180,E1 27194.884,E2 27194.884} C_VEL
LIN {X 0,Y 720.183,Z 401.52,A -85,B 0,C 180,E1 27192.201,E2 27192.201} C_VEL
LIN {X 0,Y 720.194,Z 401.502,A -85,B 0,C 180,E1 27189.107,E2 27189.107} C_VEL
LIN {X 0,Y 720.168,Z 401.518,A -85,B 0,C 180,E1 27186.377,E2 27186.377} C_VEL
LIN {X 0,Y 720.215,Z 401.507,A -85,B 0,C 180,E1 27183.582,E2 27183.582} C_VEL
LIN {X 0,Y 720.183,Z 401.513,A -85,B 0,C 180,E1 27180.636,E2 27180.636} C_VEL
LIN {X 0,Y 720.207,Z 401.514,A -85,B 0,C 180,E1 27177.772,E2 27177.772} C_VEL
LIN {X 0,Y 720.205,Z 401.511,A -85,B 0,C 180,E1 27174.663,E2 27174.663} C_VEL
LIN {X 0,Y 720.206,Z 401.515,A -85,B 0,C 180,E1 27171.698,E2 27171.698} C_VEL
LIN {X 0,Y 720.214,Z 401.51,A -85,B 0,C 180,E1 27168.564,E2 27168.564} C_VEL
LIN {X 0,Y 720.214,Z 401.512,A -85,B 0,C 180,E1 27165.528,E2 27165.528} C_VEL
LIN {X 0,Y 720.204,Z 401.513,A -85,B 0,C 180,E1 27163.625,E2 27163.625} C_VEL
LIN {X 0,Y 719.243,Z 401.642,A -85,B 0,C 180,E1 27163.012,E2 27163.012} C_VEL
LIN {X 0,Y 712.796,Z 402.44,A -85,B 0,C 180,E1 27161.296,E2 27161.296} C_VEL
LIN {X 0,Y 712.259,Z 402.498,A -85,B 0,C 180,E1 27160.85,E2 27160.85} C_VEL
LIN {X 0,Y 712.265,Z 402.499,A -85,B 0,C 180,E1 27157.987,E2 27157.987} C_VEL
LIN {X 0,Y 712.263,Z 402.497,A -85,B 0,C 180,E1 27155.004,E2 27155.004} C_VEL
LIN {X 0,Y 712.281,Z 402.5,A -85,B 0,C 180,E1 27152.004,E2 27152.004} C_VEL
LIN {X 0,Y 712.269,Z 402.503,A -85,B 0,C 180,E1 27148.989,E2 27148.989} C_VEL
LIN {X 0,Y 712.265,Z 402.494,A -85,B 0,C 180,E1 27146.033,E2 27146.033} C_VEL
LIN {X 0,Y 712.266,Z 402.502,A -85,B 0,C 180,E1 27142.88,E2 27142.88} C_VEL
LIN {X 0,Y 712.25,Z 402.506,A -85,B 0,C 180,E1 27139.987,E2 27139.987} C_VEL
LIN {X 0,Y 712.279,Z 402.511,A -85,B 0,C 180,E1 27136.981,E2 27136.981} C_VEL
LIN {X 0,Y 712.286,Z 402.541,A -85,B 0,C 180,E1 27135.421,E2 27135.421} C_VEL
LIN {X 0,Y 713.529,Z 405.91,A -85,B 0,C 180,E1 27135.067,E2 27135.067} C_VEL
LIN {X 0,Y 719.248,Z 418.345,A -85,B 0,C 180,E1 27133.734,E2 27133.734} C_VEL
LIN {X 0,Y 721.687,Z 422.643,A -85,B 0,C 180,E1 27133.491,E2 27133.491} C_VEL
LIN {X 0,Y 724.032,Z 431.845,A -85,B 0,C 180,E1 27133.192,E2 27133.192} C_VEL
LIN {X 0,Y 722.638,Z 643.066,A -85,B 0,C 180,E1 27130.531,E2 27130.531} C_VEL
LIN {X 0,Y 721.285,Z 867.911,A -85,B 0,C 180,E1 27127.791,E2 27127.791} C_VEL
LIN {X 0,Y 720.971,Z 902.736,A -85,B 0,C 180,E1 27127.331,E2 27127.331} C_VEL
LIN {X 0,Y 720.474,Z 929.904,A -85,B 0,C 180,E1 27126.808,E2 27126.808} C_VEL
LIN {X 0,Y 719.959,Z 955.344,A -85,B 0,C 180,E1 27126.166,E2 27126.166} C_VEL
LIN {X 0,Y 719.283,Z 983.248,A -85,B 0,C 180,E1 27125.282,E2 27125.282} C_VEL
LIN {X 0,Y 718.597,Z 1006.529,A -85,B 0,C 180,E1 27124.398,E2 27124.398} C_VEL
LIN {X 0,Y 717.94,Z 1027.722,A -85,B 0,C 180,E1 27123.472,E2 27123.472} C_VEL
LIN {X 0,Y 717.249,Z 1049.995,A -85,B 0,C 180,E1 27122.367,E2 27122.367} C_VEL
LIN {X 0,Y 716.464,Z 1074.881,A -85,B 0,C 180,E1 27120.95,E2 27120.95} C_VEL
LIN {X 0,Y 715.779,Z 1094.773,A -85,B 0,C 180,E1 27119.67,E2 27119.67} C_VEL
LIN {X 0,Y 715.166,Z 1113.452,A -85,B 0,C 180,E1 27118.338,E2 27118.338} C_VEL
LIN {X 0,Y 714.5,Z 1135.387,A -85,B 0,C 180,E1 27116.589,E2 27116.589} C_VEL
LIN {X 0,Y 713.953,Z 1152.89,A -85,B 0,C 180,E1 27115.022,E2 27115.022} C_VEL
LIN {X 0,Y 713.5,Z 1169.639,A -85,B 0,C 180,E1 27113.367,E2 27113.367} C_VEL
LIN {X 0,Y 713.054,Z 1187.45,A -85,B 0,C 180,E1 27111.384,E2 27111.384} C_VEL
LIN {X 0,Y 712.726,Z 1201.098,A -85,B 0,C 180,E1 27109.677,E2 27109.677} C_VEL
LIN {X 0,Y 712.49,Z 1212.682,A -85,B 0,C 180,E1 27108.07,E2 27108.07} C_VEL
LIN {X 0,Y 712.277,Z 1225.098,A -85,B 0,C 180,E1 27106.14,E2 27106.14} C_VEL
LIN {X 0,Y 712.113,Z 1237.012,A -85,B 0,C 180,E1 27103.977,E2 27103.977} C_VEL
LIN {X 0,Y 712.018,Z 1245.403,A -85,B 0,C 180,E1 27102.204,E2 27102.204} C_VEL
LIN {X 0,Y 711.976,Z 1252.259,A -85,B 0,C 180,E1 27100.521,E2 27100.521} C_VEL
LIN {X 0,Y 711.92,Z 1258.158,A -85,B 0,C 180,E1 27098.808,E2 27098.808} C_VEL
LIN {X 0,Y 711.923,Z 1263.452,A -85,B 0,C 180,E1 27096.939,E2 27096.939} C_VEL
LIN {X 0,Y 711.91,Z 1267.98,A -85,B 0,C 180,E1 27094.755,E2 27094.755} C_VEL
LIN {X 0,Y 711.909,Z 1270.636,A -85,B 0,C 180,E1 27092.659,E2 27092.659} C_VEL
LIN {X 0,Y 711.871,Z 1271.746,A -85,B 0,C 180,E1 27090.888,E2 27090.888} C_VEL
LIN {X 0,Y 711.862,Z 1271.818,A -85,B 0,C 180,E1 27089.278,E2 27089.278} C_VEL
LIN {X 0,Y 711.903,Z 1270.918,A -85,B 0,C 180,E1 27087.588,E2 27087.588} C_VEL
LIN {X 0,Y 711.916,Z 1268.751,A -85,B 0,C 180,E1 27085.653,E2 27085.653} C_VEL
LIN {X 0,Y 711.924,Z 1264.658,A -85,B 0,C 180,E1 27083.47,E2 27083.47} C_VEL
LIN {X 0,Y 711.946,Z 1258.968,A -85,B 0,C 180,E1 27081.36,E2 27081.36} C_VEL
LIN {X 0,Y 711.978,Z 1252.92,A -85,B 0,C 180,E1 27079.565,E2 27079.565} C_VEL
LIN {X 0,Y 712.01,Z 1246.355,A -85,B 0,C 180,E1 27077.925,E2 27077.925} C_VEL
LIN {X 0,Y 712.064,Z 1238.713,A -85,B 0,C 180,E1 27076.275,E2 27076.275} C_VEL
LIN {X 0,Y 712.197,Z 1230.359,A -85,B 0,C 180,E1 27074.692,E2 27074.692} C_VEL
LIN {X 0,Y 712.382,Z 1219.95,A -85,B 0,C 180,E1 27072.945,E2 27072.945} C_VEL
LIN {X 0,Y 712.659,Z 1205.665,A -85,B 0,C 180,E1 27070.837,E2 27070.837} C_VEL
LIN {X 0,Y 712.96,Z 1191.076,A -85,B 0,C 180,E1 27068.963,E2 27068.963} C_VEL
LIN {X 0,Y 713.288,Z 1176.934,A -85,B 0,C 180,E1 27067.329,E2 27067.329} C_VEL
LIN {X 0,Y 713.802,Z 1158.998,A -85,B 0,C 180,E1 27065.463,E2 27065.463} C_VEL
LIN {X 0,Y 714.33,Z 1140.351,A -85,B 0,C 180,E1 27063.752,E2 27063.752} C_VEL
LIN {X 0,Y 714.879,Z 1123.326,A -85,B 0,C 180,E1 27062.335,E2 27062.335} C_VEL
LIN {X 0,Y 715.573,Z 1101.895,A -85,B 0,C 180,E1 27060.725,E2 27060.725} C_VEL
LIN {X 0,Y 716.231,Z 1080.582,A -85,B 0,C 180,E1 27059.313,E2 27059.313} C_VEL
LIN {X 0,Y 716.901,Z 1060.967,A -85,B 0,C 180,E1 27058.147,E2 27058.147} C_VEL
LIN {X 0,Y 717.664,Z 1038.399,A -85,B 0,C 180,E1 27056.948,E2 27056.948} C_VEL
LIN {X 0,Y 718.416,Z 1012.206,A -85,B 0,C 180,E1 27055.747,E2 27055.747} C_VEL
LIN {X 0,Y 719.003,Z 990.866,A -85,B 0,C 180,E1 27054.902,E2 27054.902} C_VEL
LIN {X 0,Y 719.584,Z 968.915,A -85,B 0,C 180,E1 27054.153,E2 27054.153} C_VEL
LIN {X 0,Y 720.198,Z 944.658,A -85,B 0,C 180,E1 27053.457,E2 27053.457} C_VEL
LIN {X 0,Y 720.711,Z 917.661,A -85,B 0,C 180,E1 27052.846,E2 27052.846} C_VEL
LIN {X 0,Y 721.091,Z 891.648,A -85,B 0,C 180,E1 27052.415,E2 27052.415} C_VEL
LIN {X 0,Y 722.526,Z 660.11,A -85,B 0,C 180,E1 27049.59,E2 27049.59} C_VEL
LIN {X 0,Y 723.847,Z 455.129,A -85,B 0,C 180,E1 27047.014,E2 27047.014} C_VEL
LIN {X 0,Y 723.861,Z 430.495,A -85,B 0,C 180,E1 27046.687,E2 27046.687} C_VEL
LIN {X 0,Y 721.177,Z 421.443,A -85,B 0,C 180,E1 27046.364,E2 27046.364} C_VEL
LIN {X 0,Y 718.745,Z 417.505,A -85,B 0,C 180,E1 27046.106,E2 27046.106} C_VEL
LIN {X 0,Y 713.446,Z 405.776,A -85,B 0,C 180,E1 27044.826,E2 27044.826} C_VEL
LIN {X 0,Y 712.278,Z 402.509,A -85,B 0,C 180,E1 27044.467,E2 27044.467} C_VEL
LIN {X 0,Y 712.213,Z 402.502,A -85,B 0,C 180,E1 27041.685,E2 27041.685} C_VEL
LIN {X 0,Y 712.234,Z 402.513,A -85,B 0,C 180,E1 27039.076,E2 27039.076} C_VEL
LIN {X 0,Y 712.243,Z 402.505,A -85,B 0,C 180,E1 27035.931,E2 27035.931} C_VEL
LIN {X 0,Y 712.208,Z 402.504,A -85,B 0,C 180,E1 27033.294,E2 27033.294} C_VEL
LIN {X 0,Y 712.248,Z 402.504,A -85,B 0,C 180,E1 27030.63,E2 27030.63} C_VEL
LIN {X 0,Y 712.234,Z 402.505,A -85,B 0,C 180,E1 27027.599,E2 27027.599} C_VEL
LIN {X 0,Y 712.205,Z 402.497,A -85,B 0,C 180,E1 27024.998,E2 27024.998} C_VEL
LIN {X 0,Y 712.24,Z 402.512,A -85,B 0,C 180,E1 27022.362,E2 27022.362} C_VEL
LIN {X 0,Y 712.227,Z 402.502,A -85,B 0,C 180,E1 27019.264,E2 27019.264} C_VEL
LIN {X 0,Y 712.202,Z 402.508,A -85,B 0,C 180,E1 27016.727,E2 27016.727} C_VEL
LIN {X 0,Y 712.228,Z 402.497,A -85,B 0,C 180,E1 27014.139,E2 27014.139} C_VEL
LIN {X 0,Y 712.227,Z 402.504,A -85,B 0,C 180,E1 27011.007,E2 27011.007} C_VEL
LIN {X 0,Y 712.198,Z 402.496,A -85,B 0,C 180,E1 27008.477,E2 27008.477} C_VEL
LIN {X 0,Y 712.208,Z 402.51,A -85,B 0,C 180,E1 27006.044,E2 27006.044} C_VEL
LIN {X 0,Y 712.27,Z 402.493,A -85,B 0,C 180,E1 27003.058,E2 27003.058} C_VEL
LIN {X 0,Y 712.199,Z 402.508,A -85,B 0,C 180,E1 27000.322,E2 27000.322} C_VEL
LIN {X 0,Y 712.196,Z 402.506,A -85,B 0,C 180,E1 26997.908,E2 26997.908} C_VEL
LIN {X 0,Y 712.263,Z 402.502,A -85,B 0,C 180,E1 26995.168,E2 26995.168} C_VEL
LIN {X 0,Y 712.209,Z 402.504,A -85,B 0,C 180,E1 26992.254,E2 26992.254} C_VEL
LIN {X 0,Y 712.19,Z 402.501,A -85,B 0,C 180,E1 26989.766,E2 26989.766} C_VEL
LIN {X 0,Y 712.209,Z 402.511,A -85,B 0,C 180,E1 26987.266,E2 26987.266} C_VEL
LIN {X 0,Y 712.233,Z 402.503,A -85,B 0,C 180,E1 26984.196,E2 26984.196} C_VEL
LIN {X 0,Y 712.188,Z 402.509,A -85,B 0,C 180,E1 26981.585,E2 26981.585} C_VEL
LIN {X 0,Y 712.189,Z 402.497,A -85,B 0,C 180,E1 26979.194,E2 26979.194} C_VEL
LIN {X 0,Y 712.272,Z 402.509,A -85,B 0,C 180,E1 26976.416,E2 26976.416} C_VEL
LIN {X 0,Y 712.192,Z 402.508,A -85,B 0,C 180,E1 26973.483,E2 26973.483} C_VEL
LIN {X 0,Y 712.182,Z 402.509,A -85,B 0,C 180,E1 26971.12,E2 26971.12} C_VEL
LIN {X 0,Y 712.187,Z 402.508,A -85,B 0,C 180,E1 26968.797,E2 26968.797} C_VEL
LIN {X 0,Y 712.28,Z 402.498,A -85,B 0,C 180,E1 26965.936,E2 26965.936} C_VEL
LIN {X 0,Y 712.185,Z 402.512,A -85,B 0,C 180,E1 26963.065,E2 26963.065} C_VEL
LIN {X 0,Y 712.177,Z 402.515,A -85,B 0,C 180,E1 26960.671,E2 26960.671} C_VEL
LIN {X 0,Y 712.191,Z 402.506,A -85,B 0,C 180,E1 26958.281,E2 26958.281} C_VEL
LIN {X 0,Y 712.195,Z 402.535,A -85,B 0,C 180,E1 26956.183,E2 26956.183} C_VEL
LIN {X 0,Y 713.384,Z 405.757,A -85,B 0,C 180,E1 26955.845,E2 26955.845} C_VEL
LIN {X 0,Y 714.46,Z 407.969,A -85,B 0,C 180,E1 26955.593,E2 26955.593} C_VEL
LIN {X 0,Y 720.591,Z 421.817,A -85,B 0,C 180,E1 26954.103,E2 26954.103} C_VEL
LIN {X 0,Y 720.581,Z 428.201,A -85,B 0,C 180,E1 26953.68,E2 26953.68} C_VEL
LIN {X 0,Y 723.986,Z 441.386,A -85,B 0,C 180,E1 26953.247,E2 26953.247} C_VEL
LIN {X 0,Y 722.719,Z 641.179,A -85,B 0,C 180,E1 26950.723,E2 26950.723} C_VEL
LIN {X 0,Y 721.354,Z 866.558,A -85,B 0,C 180,E1 26947.972,E2 26947.972} C_VEL
LIN {X 0,Y 720.994,Z 910.103,A -85,B 0,C 180,E1 26947.417,E2 26947.417} C_VEL
LIN {X 0,Y 720.526,Z 937.469,A -85,B 0,C 180,E1 26946.906,E2 26946.906} C_VEL
LIN {X 0,Y 720.007,Z 962.922,A -85,B 0,C 180,E1 26946.278,E2 26946.278} C_VEL
LIN {X 0,Y 719.419,Z 988.579,A -85,B 0,C 180,E1 26945.488,E2 26945.488} C_VEL
LIN {X 0,Y 718.641,Z 1015.46,A -85,B 0,C 180,E1 26944.487,E2 26944.487} C_VEL
LIN {X 0,Y 717.975,Z 1036.782,A -85,B 0,C 180,E1 26943.56,E2 26943.56} C_VEL
LIN {X 0,Y 717.287,Z 1058.249,A -85,B 0,C 180,E1 26942.503,E2 26942.503} C_VEL
LIN {X 0,Y 716.519,Z 1083.474,A -85,B 0,C 180,E1 26941.082,E2 26941.082} C_VEL
LIN {X 0,Y 715.812,Z 1103.96,A -85,B 0,C 180,E1 26939.77,E2 26939.77} C_VEL
LIN {X 0,Y 715.21,Z 1122.306,A -85,B 0,C 180,E1 26938.468,E2 26938.468} C_VEL
LIN {X 0,Y 714.569,Z 1143.216,A -85,B 0,C 180,E1 26936.823,E2 26936.823} C_VEL
LIN {X 0,Y 713.986,Z 1162.019,A -85,B 0,C 180,E1 26935.149,E2 26935.149} C_VEL
LIN {X 0,Y 713.531,Z 1177.95,A -85,B 0,C 180,E1 26933.584,E2 26933.584} C_VEL
LIN {X 0,Y 713.098,Z 1195.866,A -85,B 0,C 180,E1 26931.62,E2 26931.62} C_VEL
LIN {X 0,Y 712.742,Z 1210.185,A -85,B 0,C 180,E1 26929.843,E2 26929.843} C_VEL
LIN {X 0,Y 712.505,Z 1222.213,A -85,B 0,C 180,E1 26928.182,E2 26928.182} C_VEL
LIN {X 0,Y 712.294,Z 1233.85,A -85,B 0,C 180,E1 26926.386,E2 26926.386} C_VEL
LIN {X 0,Y 712.134,Z 1246.437,A -85,B 0,C 180,E1 26924.138,E2 26924.138} C_VEL
LIN {X 0,Y 712.031,Z 1255.087,A -85,B 0,C 180,E1 26922.322,E2 26922.322} C_VEL
LIN {X 0,Y 711.972,Z 1262.139,A -85,B 0,C 180,E1 26920.599,E2 26920.599} C_VEL
LIN {X 0,Y 711.916,Z 1268.058,A -85,B 0,C 180,E1 26918.885,E2 26918.885} C_VEL
LIN {X 0,Y 711.925,Z 1273.376,A -85,B 0,C 180,E1 26917.016,E2 26917.016} C_VEL
LIN {X 0,Y 711.914,Z 1277.932,A -85,B 0,C 180,E1 26914.832,E2 26914.832} C_VEL
LIN {X 0,Y 711.911,Z 1280.611,A -85,B 0,C 180,E1 26912.735,E2 26912.735} C_VEL
LIN {X 0,Y 711.871,Z 1281.738,A -85,B 0,C 180,E1 26910.963,E2 26910.963} C_VEL
LIN {X 0,Y 711.863,Z 1281.826,A -85,B 0,C 180,E1 26909.354,E2 26909.354} C_VEL
LIN {X 0,Y 711.906,Z 1280.944,A -85,B 0,C 180,E1 26907.663,E2 26907.663} C_VEL
LIN {X 0,Y 711.919,Z 1278.799,A -85,B 0,C 180,E1 26905.729,E2 26905.729} C_VEL
LIN {X 0,Y 711.927,Z 1274.73,A -85,B 0,C 180,E1 26903.547,E2 26903.547} C_VEL
LIN {X 0,Y 711.946,Z 1269.068,A -85,B 0,C 180,E1 26901.437,E2 26901.437} C_VEL
LIN {X 0,Y 711.981,Z 1263.039,A -85,B 0,C 180,E1 26899.642,E2 26899.642} C_VEL
LIN {X 0,Y 712.009,Z 1256.138,A -85,B 0,C 180,E1 26897.92,E2 26897.92} C_VEL
LIN {X 0,Y 712.062,Z 1248.824,A -85,B 0,C 180,E1 26896.342,E2 26896.342} C_VEL
LIN {X 0,Y 712.194,Z 1240.588,A -85,B 0,C 180,E1 26894.778,E2 26894.778} C_VEL
LIN {X 0,Y 712.371,Z 1230.686,A -85,B 0,C 180,E1 26893.108,E2 26893.108} C_VEL
LIN {X 0,Y 712.639,Z 1217.169,A -85,B 0,C 180,E1 26891.087,E2 26891.087} C_VEL
LIN {X 0,Y 712.945,Z 1201.641,A -85,B 0,C 180,E1 26889.076,E2 26889.076} C_VEL
LIN {X 0,Y 713.256,Z 1188.013,A -85,B 0,C 180,E1 26887.493,E2 26887.493} C_VEL
LIN {X 0,Y 713.712,Z 1172.401,A -85,B 0,C 180,E1 26885.851,E2 26885.851} C_VEL
LIN {X 0,Y 714.249,Z 1152.638,A -85,B 0,C 180,E1 26883.995,E2 26883.995} C_VEL
LIN {X 0,Y 714.802,Z 1135.479,A -85,B 0,C 180,E1 26882.553,E2 26882.553} C_VEL
LIN {X 0,Y 715.402,Z 1116.789,A -85,B 0,C 180,E1 26881.124,E2 26881.124} C_VEL
LIN {X 0,Y 716.163,Z 1092.527,A -85,B 0,C 180,E1 26879.479,E2 26879.479} C_VEL
LIN {X 0,Y 716.841,Z 1072.403,A -85,B 0,C 180,E1 26878.273,E2 26878.273} C_VEL
LIN {X 0,Y 717.526,Z 1051.906,A -85,B 0,C 180,E1 26877.172,E2 26877.172} C_VEL
LIN {X 0,Y 718.348,Z 1026.514,A -85,B 0,C 180,E1 26875.974,E2 26875.974} C_VEL
LIN {X 0,Y 718.977,Z 1002.23,A -85,B 0,C 180,E1 26874.998,E2 26874.998} C_VEL
LIN {X 0,Y 719.54,Z 980.455,A -85,B 0,C 180,E1 26874.247,E2 26874.247} C_VEL
LIN {X 0,Y 720.134,Z 957.158,A -85,B 0,C 180,E1 26873.567,E2 26873.567} C_VEL
LIN {X 0,Y 720.672,Z 930.198,A -85,B 0,C 180,E1 26872.941,E2 26872.941} C_VEL
LIN {X 0,Y 721.072,Z 903.176,A -85,B 0,C 180,E1 26872.481,E2 26872.481} C_VEL
LIN {X 0,Y 722.518,Z 671.462,A -85,B 0,C 180,E1 26869.652,E2 26869.652} C_VEL
LIN {X 0,Y 723.775,Z 472.851,A -85,B 0,C 180,E1 26867.156,E2 26867.156} C_VEL
LIN {X 0,Y 723.842,Z 440.108,A -85,B 0,C 180,E1 26866.726,E2 26866.726} C_VEL
LIN {X 0,Y 720.47,Z 427.342,A -85,B 0,C 180,E1 26866.279,E2 26866.279} C_VEL
LIN {X 0,Y 720.438,Z 421.118,A -85,B 0,C 180,E1 26865.835,E2 26865.835} C_VEL
LIN {X 0,Y 713.801,Z 406.364,A -85,B 0,C 180,E1 26864.235,E2 26864.235} C_VEL
LIN {X 0,Y 712.241,Z 402.894,A -85,B 0,C 180,E1 26863.847,E2 26863.847} C_VEL
LIN {X 0,Y 712.182,Z 402.52,A -85,B 0,C 180,E1 26863.802,E2 26863.802} C_VEL
LIN {X 0,Y 712.173,Z 402.506,A -85,B 0,C 180,E1 26861.398,E2 26861.398} C_VEL
LIN {X 0,Y 712.186,Z 402.516,A -85,B 0,C 180,E1 26859.068,E2 26859.068} C_VEL
LIN {X 0,Y 712.265,Z 402.51,A -85,B 0,C 180,E1 26856.129,E2 26856.129} C_VEL
LIN {X 0,Y 712.19,Z 402.507,A -85,B 0,C 180,E1 26853.392,E2 26853.392} C_VEL
LIN {X 0,Y 712.193,Z 402.51,A -85,B 0,C 180,E1 26851.015,E2 26851.015} C_VEL
LIN {X 0,Y 712.259,Z 402.507,A -85,B 0,C 180,E1 26848.327,E2 26848.327} C_VEL
LIN {X 0,Y 712.215,Z 402.496,A -85,B 0,C 180,E1 26845.353,E2 26845.353} C_VEL
LIN {X 0,Y 712.204,Z 402.509,A -85,B 0,C 180,E1 26842.886,E2 26842.886} C_VEL
LIN {X 0,Y 712.256,Z 402.499,A -85,B 0,C 180,E1 26840.203,E2 26840.203} C_VEL
LIN {X 0,Y 712.228,Z 402.505,A -85,B 0,C 180,E1 26837.147,E2 26837.147} C_VEL
LIN {X 0,Y 712.217,Z 402.496,A -85,B 0,C 180,E1 26834.555,E2 26834.555} C_VEL
LIN {X 0,Y 712.281,Z 402.507,A -85,B 0,C 180,E1 26831.745,E2 26831.745} C_VEL
LIN {X 0,Y 712.23,Z 402.492,A -85,B 0,C 180,E1 26828.802,E2 26828.802} C_VEL
LIN {X 0,Y 712.25,Z 402.51,A -85,B 0,C 180,E1 26826.044,E2 26826.044} C_VEL
LIN {X 0,Y 712.257,Z 402.489,A -85,B 0,C 180,E1 26822.897,E2 26822.897} C_VEL
LIN {X 0,Y 712.245,Z 402.508,A -85,B 0,C 180,E1 26820.08,E2 26820.08} C_VEL
LIN {X 0,Y 712.274,Z 402.49,A -85,B 0,C 180,E1 26817.103,E2 26817.103} C_VEL
LIN {X 0,Y 712.244,Z 402.505,A -85,B 0,C 180,E1 26814.199,E2 26814.199} C_VEL
LIN {X 0,Y 712.273,Z 402.495,A -85,B 0,C 180,E1 26811.361,E2 26811.361} C_VEL
LIN {X 0,Y 712.26,Z 402.501,A -85,B 0,C 180,E1 26808.337,E2 26808.337} C_VEL
LIN {X 0,Y 712.276,Z 402.496,A -85,B 0,C 180,E1 26805.364,E2 26805.364} C_VEL
LIN {X 0,Y 712.278,Z 402.499,A -85,B 0,C 180,E1 26802.349,E2 26802.349} C_VEL
LIN {X 0,Y 712.259,Z 402.498,A -85,B 0,C 180,E1 26800.85,E2 26800.85} C_VEL
LIN {X 0,Y 711.278,Z 402.617,A -85,B 0,C 180,E1 26800.23,E2 26800.23} C_VEL
LIN {X 0,Y 704.876,Z 403.419,A -85,B 0,C 180,E1 26798.494,E2 26798.494} C_VEL
LIN {X 0,Y 704.329,Z 403.487,A -85,B 0,C 180,E1 26798.043,E2 26798.043} C_VEL
LIN {X 0,Y 704.328,Z 403.484,A -85,B 0,C 180,E1 26795.062,E2 26795.062} C_VEL
LIN {X 0,Y 704.343,Z 403.489,A -85,B 0,C 180,E1 26792.005,E2 26792.005} C_VEL
LIN {X 0,Y 704.329,Z 403.491,A -85,B 0,C 180,E1 26788.98,E2 26788.98} C_VEL
LIN {X 0,Y 704.33,Z 403.482,A -85,B 0,C 180,E1 26785.99,E2 26785.99} C_VEL
LIN {X 0,Y 704.328,Z 403.49,A -85,B 0,C 180,E1 26782.89,E2 26782.89} C_VEL
LIN {X 0,Y 704.317,Z 403.495,A -85,B 0,C 180,E1 26779.925,E2 26779.925} C_VEL
LIN {X 0,Y 704.33,Z 403.5,A -85,B 0,C 180,E1 26776.822,E2 26776.822} C_VEL
LIN {X 0,Y 704.312,Z 403.595,A -85,B 0,C 180,E1 26776.003,E2 26776.003} C_VEL
LIN {X 0,Y 705.445,Z 406.688,A -85,B 0,C 180,E1 26775.671,E2 26775.671} C_VEL
LIN {X 0,Y 710.811,Z 418.35,A -85,B 0,C 180,E1 26774.389,E2 26774.389} C_VEL
LIN {X 0,Y 716.437,Z 427.011,A -85,B 0,C 180,E1 26773.832,E2 26773.832} C_VEL
LIN {X 0,Y 718.174,Z 434.001,A -85,B 0,C 180,E1 26773.604,E2 26773.604} C_VEL
LIN {X 0,Y 716.537,Z 645.025,A -85,B 0,C 180,E1 26770.924,E2 26770.924} C_VEL
LIN {X 0,Y 714.949,Z 869.462,A -85,B 0,C 180,E1 26768.167,E2 26768.167} C_VEL
LIN {X 0,Y 714.58,Z 903.287,A -85,B 0,C 180,E1 26767.713,E2 26767.713} C_VEL
LIN {X 0,Y 714.004,Z 930.298,A -85,B 0,C 180,E1 26767.188,E2 26767.188} C_VEL
LIN {X 0,Y 713.409,Z 955.572,A -85,B 0,C 180,E1 26766.545,E2 26766.545} C_VEL
LIN {X 0,Y 712.602,Z 983.803,A -85,B 0,C 180,E1 26765.643,E2 26765.643} C_VEL
LIN {X 0,Y 711.836,Z 1006.547,A -85,B 0,C 180,E1 26764.772,E2 26764.772} C_VEL
LIN {X 0,Y 711.07,Z 1027.738,A -85,B 0,C 180,E1 26763.839,E2 26763.839} C_VEL
LIN {X 0,Y 710.236,Z 1050.01,A -85,B 0,C 180,E1 26762.726,E2 26762.726} C_VEL
LIN {X 0,Y 709.314,Z 1074.887,A -85,B 0,C 180,E1 26761.297,E2 26761.297} C_VEL
LIN {X 0,Y 708.528,Z 1094.57,A -85,B 0,C 180,E1 26760.019,E2 26760.019} C_VEL
LIN {X 0,Y 707.815,Z 1113.108,A -85,B 0,C 180,E1 26758.687,E2 26758.687} C_VEL
LIN {X 0,Y 707.01,Z 1134.709,A -85,B 0,C 180,E1 26756.955,E2 26756.955} C_VEL
LIN {X 0,Y 706.388,Z 1152.431,A -85,B 0,C 180,E1 26755.354,E2 26755.354} C_VEL
LIN {X 0,Y 705.831,Z 1168.797,A -85,B 0,C 180,E1 26753.725,E2 26753.725} C_VEL
LIN {X 0,Y 705.276,Z 1187.457,A -85,B 0,C 180,E1 26751.631,E2 26751.631} C_VEL
LIN {X 0,Y 704.886,Z 1201.104,A -85,B 0,C 180,E1 26749.905,E2 26749.905} C_VEL
LIN {X 0,Y 704.606,Z 1213.27,A -85,B 0,C 180,E1 26748.193,E2 26748.193} C_VEL
LIN {X 0,Y 704.334,Z 1226.619,A -85,B 0,C 180,E1 26746.073,E2 26746.073} C_VEL
LIN {X 0,Y 704.157,Z 1237.426,A -85,B 0,C 180,E1 26744.055,E2 26744.055} C_VEL
LIN {X 0,Y 704.046,Z 1245.667,A -85,B 0,C 180,E1 26742.284,E2 26742.284} C_VEL
LIN {X 0,Y 703.986,Z 1252.344,A -85,B 0,C 180,E1 26740.62,E2 26740.62} C_VEL
LIN {X 0,Y 703.918,Z 1258.16,A -85,B 0,C 180,E1 26738.909,E2 26738.909} C_VEL
LIN {X 0,Y 703.929,Z 1263.453,A -85,B 0,C 180,E1 26737.019,E2 26737.019} C_VEL
LIN {X 0,Y 703.913,Z 1267.981,A -85,B 0,C 180,E1 26734.81,E2 26734.81} C_VEL
LIN {X 0,Y 703.91,Z 1270.637,A -85,B 0,C 180,E1 26732.689,E2 26732.689} C_VEL
LIN {X 0,Y 703.872,Z 1271.747,A -85,B 0,C 180,E1 26730.898,E2 26730.898} C_VEL
LIN {X 0,Y 703.862,Z 1271.818,A -85,B 0,C 180,E1 26729.27,E2 26729.27} C_VEL
LIN {X 0,Y 703.903,Z 1270.918,A -85,B 0,C 180,E1 26727.56,E2 26727.56} C_VEL
LIN {X 0,Y 703.914,Z 1268.751,A -85,B 0,C 180,E1 26725.603,E2 26725.603} C_VEL
LIN {X 0,Y 703.924,Z 1264.657,A -85,B 0,C 180,E1 26723.396,E2 26723.396} C_VEL
LIN {X 0,Y 703.943,Z 1258.967,A -85,B 0,C 180,E1 26721.261,E2 26721.261} C_VEL
LIN {X 0,Y 703.985,Z 1252.919,A -85,B 0,C 180,E1 26719.445,E2 26719.445} C_VEL
LIN {X 0,Y 704.037,Z 1246.354,A -85,B 0,C 180,E1 26717.786,E2 26717.786} C_VEL
LIN {X 0,Y 704.112,Z 1238.711,A -85,B 0,C 180,E1 26716.117,E2 26716.117} C_VEL
LIN {X 0,Y 704.284,Z 1229.932,A -85,B 0,C 180,E1 26714.438,E2 26714.438} C_VEL
LIN {X 0,Y 704.484,Z 1218.514,A -85,B 0,C 180,E1 26712.514,E2 26712.514} C_VEL
LIN {X 0,Y 704.836,Z 1203.747,A -85,B 0,C 180,E1 26710.357,E2 26710.357} C_VEL
LIN {X 0,Y 705.191,Z 1190.362,A -85,B 0,C 180,E1 26708.633,E2 26708.633} C_VEL
LIN {X 0,Y 705.633,Z 1175.371,A -85,B 0,C 180,E1 26706.893,E2 26706.893} C_VEL
LIN {X 0,Y 706.25,Z 1155.749,A -85,B 0,C 180,E1 26704.87,E2 26704.87} C_VEL
LIN {X 0,Y 706.865,Z 1138.884,A -85,B 0,C 180,E1 26703.323,E2 26703.323} C_VEL
LIN {X 0,Y 707.575,Z 1119.989,A -85,B 0,C 180,E1 26701.749,E2 26701.749} C_VEL
LIN {X 0,Y 708.392,Z 1097.913,A -85,B 0,C 180,E1 26700.12,E2 26700.12} C_VEL
LIN {X 0,Y 709.151,Z 1078.556,A -85,B 0,C 180,E1 26698.842,E2 26698.842} C_VEL
LIN {X 0,Y 709.949,Z 1058.431,A -85,B 0,C 180,E1 26697.648,E2 26697.648} C_VEL
LIN {X 0,Y 710.891,Z 1032.676,A -85,B 0,C 180,E1 26696.302,E2 26696.302} C_VEL
LIN {X 0,Y 711.693,Z 1009.847,A -85,B 0,C 180,E1 26695.275,E2 26695.275} C_VEL
LIN {X 0,Y 712.416,Z 988.309,A -85,B 0,C 180,E1 26694.431,E2 26694.431} C_VEL
LIN {X 0,Y 713.136,Z 964.461,A -85,B 0,C 180,E1 26693.628,E2 26693.628} C_VEL
LIN {X 0,Y 713.855,Z 937.713,A -85,B 0,C 180,E1 26692.895,E2 26692.895} C_VEL
LIN {X 0,Y 714.402,Z 912.069,A -85,B 0,C 180,E1 26692.352,E2 26692.352} C_VEL
LIN {X 0,Y 714.808,Z 885.982,A -85,B 0,C 180,E1 26691.946,E2 26691.946} C_VEL
LIN {X 0,Y 716.429,Z 659.125,A -85,B 0,C 180,E1 26689.161,E2 26689.161} C_VEL
LIN {X 0,Y 717.987,Z 454.295,A -85,B 0,C 180,E1 26686.566,E2 26686.566} C_VEL
LIN {X 0,Y 718.005,Z 432.708,A -85,B 0,C 180,E1 26686.276,E2 26686.276} C_VEL
LIN {X 0,Y 715.992,Z 426.149,A -85,B 0,C 180,E1 26686.032,E2 26686.032} C_VEL
LIN {X 0,Y 710.403,Z 417.709,A -85,B 0,C 180,E1 26685.471,E2 26685.471} C_VEL
LIN {X 0,Y 705.766,Z 407.183,A -85,B 0,C 180,E1 26684.303,E2 26684.303} C_VEL
LIN {X 0,Y 704.31,Z 403.708,A -85,B 0,C 180,E1 26683.915,E2 26683.915} C_VEL
LIN {X 0,Y 704.276,Z 403.488,A -85,B 0,C 180,E1 26681.422,E2 26681.422} C_VEL
LIN {X 0,Y 704.346,Z 403.497,A -85,B 0,C 180,E1 26678.545,E2 26678.545} C_VEL
LIN {X 0,Y 704.277,Z 403.496,A -85,B 0,C 180,E1 26675.598,E2 26675.598} C_VEL
LIN {X 0,Y 704.279,Z 403.494,A -85,B 0,C 180,E1 26673.037,E2 26673.037} C_VEL
LIN {X 0,Y 704.346,Z 403.482,A -85,B 0,C 180,E1 26670.074,E2 26670.074} C_VEL
LIN {X 0,Y 704.272,Z 403.496,A -85,B 0,C 180,E1 26667.292,E2 26667.292} C_VEL
LIN {X 0,Y 704.277,Z 403.486,A -85,B 0,C 180,E1 26664.695,E2 26664.695} C_VEL
LIN {X 0,Y 704.341,Z 403.487,A -85,B 0,C 180,E1 26661.748,E2 26661.748} C_VEL
LIN {X 0,Y 704.268,Z 403.492,A -85,B 0,C 180,E1 26658.973,E2 26658.973} C_VEL
LIN {X 0,Y 704.269,Z 403.498,A -85,B 0,C 180,E1 26656.496,E2 26656.496} C_VEL
LIN {X 0,Y 704.345,Z 403.488,A -85,B 0,C 180,E1 26653.63,E2 26653.63} C_VEL
LIN {X 0,Y 704.266,Z 403.494,A -85,B 0,C 180,E1 26650.719,E2 26650.719} C_VEL
LIN {X 0,Y 704.263,Z 403.484,A -85,B 0,C 180,E1 26648.244,E2 26648.244} C_VEL
LIN {X 0,Y 704.339,Z 403.498,A -85,B 0,C 180,E1 26645.458,E2 26645.458} C_VEL
LIN {X 0,Y 704.266,Z 403.484,A -85,B 0,C 180,E1 26642.523,E2 26642.523} C_VEL
LIN {X 0,Y 704.257,Z 403.498,A -85,B 0,C 180,E1 26640.081,E2 26640.081} C_VEL
LIN {X 0,Y 704.292,Z 403.494,A -85,B 0,C 180,E1 26637.478,E2 26637.478} C_VEL
LIN {X 0,Y 704.275,Z 403.497,A -85,B 0,C 180,E1 26634.355,E2 26634.355} C_VEL
LIN {X 0,Y 704.252,Z 403.493,A -85,B 0,C 180,E1 26631.838,E2 26631.838} C_VEL
LIN {X 0,Y 704.269,Z 403.49,A -85,B 0,C 180,E1 26629.364,E2 26629.364} C_VEL
LIN {X 0,Y 704.297,Z 403.489,A -85,B 0,C 180,E1 26626.285,E2 26626.285} C_VEL
LIN {X 0,Y 704.251,Z 403.493,A -85,B 0,C 180,E1 26623.673,E2 26623.673} C_VEL
LIN {X 0,Y 704.254,Z 403.499,A -85,B 0,C 180,E1 26621.246,E2 26621.246} C_VEL
LIN {X 0,Y 704.341,Z 403.487,A -85,B 0,C 180,E1 26618.397,E2 26618.397} C_VEL
LIN {X 0,Y 704.252,Z 403.493,A -85,B 0,C 180,E1 26615.505,E2 26615.505} C_VEL
LIN {X 0,Y 704.246,Z 403.497,A -85,B 0,C 180,E1 26613.069,E2 26613.069} C_VEL
LIN {X 0,Y 704.273,Z 403.499,A -85,B 0,C 180,E1 26610.578,E2 26610.578} C_VEL
LIN {X 0,Y 704.267,Z 403.499,A -85,B 0,C 180,E1 26607.446,E2 26607.446} C_VEL
LIN {X 0,Y 704.242,Z 403.498,A -85,B 0,C 180,E1 26604.998,E2 26604.998} C_VEL
LIN {X 0,Y 704.242,Z 403.502,A -85,B 0,C 180,E1 26602.657,E2 26602.657} C_VEL
LIN {X 0,Y 704.302,Z 403.499,A -85,B 0,C 180,E1 26599.975,E2 26599.975} C_VEL
LIN {X 0,Y 704.254,Z 403.508,A -85,B 0,C 180,E1 26596.98,E2 26596.98} C_VEL
LIN {X 0,Y 704.263,Z 403.671,A -85,B 0,C 180,E1 26596.773,E2 26596.773} C_VEL
LIN {X 0,Y 705.696,Z 407.203,A -85,B 0,C 180,E1 26596.382,E2 26596.382} C_VEL
LIN {X 0,Y 710.253,Z 417.161,A -85,B 0,C 180,E1 26595.259,E2 26595.259} C_VEL
LIN {X 0,Y 714.085,Z 425.941,A -85,B 0,C 180,E1 26594.314,E2 26594.314} C_VEL
LIN {X 0,Y 714.213,Z 428.444,A -85,B 0,C 180,E1 26594.166,E2 26594.166} C_VEL
LIN {X 0,Y 718.131,Z 443.546,A -85,B 0,C 180,E1 26593.658,E2 26593.658} C_VEL
LIN {X 0,Y 716.627,Z 643.858,A -85,B 0,C 180,E1 26591.108,E2 26591.108} C_VEL
LIN {X 0,Y 715.019,Z 870.102,A -85,B 0,C 180,E1 26588.324,E2 26588.324} C_VEL
LIN {X 0,Y 714.609,Z 911.094,A -85,B 0,C 180,E1 26587.794,E2 26587.794} C_VEL
LIN {X 0,Y 714.052,Z 938.598,A -85,B 0,C 180,E1 26587.271,E2 26587.271} C_VEL
LIN {X 0,Y 713.45,Z 963.698,A -85,B 0,C 180,E1 26586.642,E2 26586.642} C_VEL
LIN {X 0,Y 712.731,Z 990.723,A -85,B 0,C 180,E1 26585.799,E2 26585.799} C_VEL
LIN {X 0,Y 711.882,Z 1015.457,A -85,B 0,C 180,E1 26584.861,E2 26584.861} C_VEL
LIN {X 0,Y 711.11,Z 1036.785,A -85,B 0,C 180,E1 26583.928,E2 26583.928} C_VEL
LIN {X 0,Y 710.332,Z 1057.388,A -85,B 0,C 180,E1 26582.907,E2 26582.907} C_VEL
LIN {X 0,Y 709.431,Z 1082.002,A -85,B 0,C 180,E1 26581.522,E2 26581.522} C_VEL
LIN {X 0,Y 708.562,Z 1103.869,A -85,B 0,C 180,E1 26580.112,E2 26580.112} C_VEL
LIN {X 0,Y 707.845,Z 1122.307,A -85,B 0,C 180,E1 26578.792,E2 26578.792} C_VEL
LIN {X 0,Y 707.067,Z 1143.239,A -85,B 0,C 180,E1 26577.129,E2 26577.129} C_VEL
LIN {X 0,Y 706.404,Z 1162.046,A -85,B 0,C 180,E1 26575.435,E2 26575.435} C_VEL
LIN {X 0,Y 705.84,Z 1178.427,A -85,B 0,C 180,E1 26573.808,E2 26573.808} C_VEL
LIN {X 0,Y 705.286,Z 1197.153,A -85,B 0,C 180,E1 26571.713,E2 26571.713} C_VEL
LIN {X 0,Y 704.891,Z 1210.832,A -85,B 0,C 180,E1 26569.987,E2 26569.987} C_VEL
LIN {X 0,Y 704.615,Z 1223.026,A -85,B 0,C 180,E1 26568.274,E2 26568.274} C_VEL
LIN {X 0,Y 704.34,Z 1236.423,A -85,B 0,C 180,E1 26566.152,E2 26566.152} C_VEL
LIN {X 0,Y 704.156,Z 1247.402,A -85,B 0,C 180,E1 26564.104,E2 26564.104} C_VEL
LIN {X 0,Y 704.057,Z 1255.446,A -85,B 0,C 180,E1 26562.38,E2 26562.38} C_VEL
LIN {X 0,Y 703.983,Z 1262.446,A -85,B 0,C 180,E1 26560.637,E2 26560.637} C_VEL
LIN {X 0,Y 703.916,Z 1268.058,A -85,B 0,C 180,E1 26558.987,E2 26558.987} C_VEL
LIN {X 0,Y 703.933,Z 1273.376,A -85,B 0,C 180,E1 26557.096,E2 26557.096} C_VEL
LIN {X 0,Y 703.916,Z 1277.932,A -85,B 0,C 180,E1 26554.887,E2 26554.887} C_VEL
LIN {X 0,Y 703.912,Z 1280.611,A -85,B 0,C 180,E1 26552.766,E2 26552.766} C_VEL
LIN {X 0,Y 703.871,Z 1281.738,A -85,B 0,C 180,E1 26550.974,E2 26550.974} C_VEL
LIN {X 0,Y 703.863,Z 1281.826,A -85,B 0,C 180,E1 26549.347,E2 26549.347} C_VEL
LIN {X 0,Y 703.905,Z 1280.944,A -85,B 0,C 180,E1 26547.637,E2 26547.637} C_VEL
LIN {X 0,Y 703.917,Z 1278.799,A -85,B 0,C 180,E1 26545.68,E2 26545.68} C_VEL
LIN {X 0,Y 703.927,Z 1274.73,A -85,B 0,C 180,E1 26543.473,E2 26543.473} C_VEL
LIN {X 0,Y 703.945,Z 1269.068,A -85,B 0,C 180,E1 26541.338,E2 26541.338} C_VEL
LIN {X 0,Y 703.989,Z 1263.04,A -85,B 0,C 180,E1 26539.523,E2 26539.523} C_VEL
LIN {X 0,Y 704.037,Z 1256.139,A -85,B 0,C 180,E1 26537.781,E2 26537.781} C_VEL
LIN {X 0,Y 704.118,Z 1248.468,A -85,B 0,C 180,E1 26536.112,E2 26536.112} C_VEL
LIN {X 0,Y 704.293,Z 1239.659,A -85,B 0,C 180,E1 26534.434,E2 26534.434} C_VEL
LIN {X 0,Y 704.505,Z 1227.553,A -85,B 0,C 180,E1 26532.402,E2 26532.402} C_VEL
LIN {X 0,Y 704.844,Z 1213.374,A -85,B 0,C 180,E1 26530.353,E2 26530.353} C_VEL
LIN {X 0,Y 705.204,Z 1199.954,A -85,B 0,C 180,E1 26528.628,E2 26528.628} C_VEL
LIN {X 0,Y 705.66,Z 1184.755,A -85,B 0,C 180,E1 26526.869,E2 26526.869} C_VEL
LIN {X 0,Y 706.27,Z 1165.228,A -85,B 0,C 180,E1 26524.866,E2 26524.866} C_VEL
LIN {X 0,Y 706.871,Z 1148.766,A -85,B 0,C 180,E1 26523.357,E2 26523.357} C_VEL
LIN {X 0,Y 707.578,Z 1129.936,A -85,B 0,C 180,E1 26521.79,E2 26521.79} C_VEL
LIN {X 0,Y 708.393,Z 1107.857,A -85,B 0,C 180,E1 26520.161,E2 26520.161} C_VEL
LIN {X 0,Y 709.158,Z 1088.429,A -85,B 0,C 180,E1 26518.88,E2 26518.88} C_VEL
LIN {X 0,Y 709.96,Z 1068.121,A -85,B 0,C 180,E1 26517.675,E2 26517.675} C_VEL
LIN {X 0,Y 710.89,Z 1042.634,A -85,B 0,C 180,E1 26516.345,E2 26516.345} C_VEL
LIN {X 0,Y 711.696,Z 1019.81,A -85,B 0,C 180,E1 26515.319,E2 26515.319} C_VEL
LIN {X 0,Y 712.418,Z 998.277,A -85,B 0,C 180,E1 26514.474,E2 26514.474} C_VEL
LIN {X 0,Y 713.161,Z 973.696,A -85,B 0,C 180,E1 26513.649,E2 26513.649} C_VEL
LIN {X 0,Y 713.88,Z 946.709,A -85,B 0,C 180,E1 26512.916,E2 26512.916} C_VEL
LIN {X 0,Y 714.413,Z 921.356,A -85,B 0,C 180,E1 26512.383,E2 26512.383} C_VEL
LIN {X 0,Y 714.823,Z 894.915,A -85,B 0,C 180,E1 26511.977,E2 26511.977} C_VEL
LIN {X 0,Y 716.439,Z 667.775,A -85,B 0,C 180,E1 26509.19,E2 26509.19} C_VEL
LIN {X 0,Y 717.918,Z 470.051,A -85,B 0,C 180,E1 26506.683,E2 26506.683} C_VEL
LIN {X 0,Y 717.974,Z 442.208,A -85,B 0,C 180,E1 26506.311,E2 26506.311} C_VEL
LIN {X 0,Y 714.047,Z 427.342,A -85,B 0,C 180,E1 26505.784,E2 26505.784} C_VEL
LIN {X 0,Y 713.995,Z 425.347,A -85,B 0,C 180,E1 26505.636,E2 26505.636} C_VEL
LIN {X 0,Y 707.473,Z 411.027,A -85,B 0,C 180,E1 26504.056,E2 26504.056} C_VEL
LIN {X 0,Y 705.337,Z 406.677,A -85,B 0,C 180,E1 26503.548,E2 26503.548} C_VEL
LIN {X 0,Y 704.241,Z 403.51,A -85,B 0,C 180,E1 26503.185,E2 26503.185} C_VEL
LIN {X 0,Y 704.319,Z 403.493,A -85,B 0,C 180,E1 26500.237,E2 26500.237} C_VEL
LIN {X 0,Y 704.244,Z 403.494,A -85,B 0,C 180,E1 26497.47,E2 26497.47} C_VEL
LIN {X 0,Y 704.249,Z 403.501,A -85,B 0,C 180,E1 26495.101,E2 26495.101} C_VEL
LIN {X 0,Y 704.324,Z 403.498,A -85,B 0,C 180,E1 26492.358,E2 26492.358} C_VEL
LIN {X 0,Y 704.267,Z 403.492,A -85,B 0,C 180,E1 26489.422,E2 26489.422} C_VEL
LIN {X 0,Y 704.262,Z 403.499,A -85,B 0,C 180,E1 26486.93,E2 26486.93} C_VEL
LIN {X 0,Y 704.34,Z 403.49,A -85,B 0,C 180,E1 26484.104,E2 26484.104} C_VEL
LIN {X 0,Y 704.275,Z 403.489,A -85,B 0,C 180,E1 26481.138,E2 26481.138} C_VEL
LIN {X 0,Y 704.281,Z 403.494,A -85,B 0,C 180,E1 26478.543,E2 26478.543} C_VEL
LIN {X 0,Y 704.344,Z 403.477,A -85,B 0,C 180,E1 26475.564,E2 26475.564} C_VEL
LIN {X 0,Y 704.282,Z 403.494,A -85,B 0,C 180,E1 26472.713,E2 26472.713} C_VEL
LIN {X 0,Y 704.336,Z 403.484,A -85,B 0,C 180,E1 26469.867,E2 26469.867} C_VEL
LIN {X 0,Y 704.301,Z 403.492,A -85,B 0,C 180,E1 26466.849,E2 26466.849} C_VEL
LIN {X 0,Y 704.309,Z 403.494,A -85,B 0,C 180,E1 26464.071,E2 26464.071} C_VEL
LIN {X 0,Y 704.337,Z 403.489,A -85,B 0,C 180,E1 26460.976,E2 26460.976} C_VEL
LIN {X 0,Y 704.307,Z 403.494,A -85,B 0,C 180,E1 26458.047,E2 26458.047} C_VEL
LIN {X 0,Y 704.334,Z 403.492,A -85,B 0,C 180,E1 26455.114,E2 26455.114} C_VEL
LIN {X 0,Y 704.308,Z 403.49,A -85,B 0,C 180,E1 26452.249,E2 26452.249} C_VEL
LIN {X 0,Y 704.335,Z 403.493,A -85,B 0,C 180,E1 26449.365,E2 26449.365} C_VEL
LIN {X 0,Y 704.329,Z 403.485,A -85,B 0,C 180,E1 26446.369,E2 26446.369} C_VEL
LIN {X 0,Y 704.339,Z 403.494,A -85,B 0,C 180,E1 26443.336,E2 26443.336} C_VEL
LIN {X 0,Y 704.337,Z 403.481,A -85,B 0,C 180,E1 26440.253,E2 26440.253} C_VEL
LIN {X 0,Y 704.329,Z 403.487,A -85,B 0,C 180,E1 26438.043,E2 26438.043} C_VEL
LIN {X 0,Y 703.328,Z 403.622,A -85,B 0,C 180,E1 26437.416,E2 26437.416} C_VEL
LIN {X 0,Y 696.935,Z 404.415,A -85,B 0,C 180,E1 26435.661,E2 26435.661} C_VEL
LIN {X 0,Y 696.396,Z 404.473,A -85,B 0,C 180,E1 26435.204,E2 26435.204} C_VEL
LIN {X 0,Y 696.401,Z 404.479,A -85,B 0,C 180,E1 26432.091,E2 26432.091} C_VEL
LIN {X 0,Y 696.389,Z 404.478,A -85,B 0,C 180,E1 26428.972,E2 26428.972} C_VEL
LIN {X 0,Y 696.396,Z 404.47,A -85,B 0,C 180,E1 26425.941,E2 26425.941} C_VEL
LIN {X 0,Y 696.381,Z 404.477,A -85,B 0,C 180,E1 26422.808,E2 26422.808} C_VEL
LIN {X 0,Y 696.383,Z 404.484,A -85,B 0,C 180,E1 26419.857,E2 26419.857} C_VEL
LIN {X 0,Y 696.382,Z 404.49,A -85,B 0,C 180,E1 26416.717,E2 26416.717} C_VEL
LIN {X 0,Y 696.4,Z 404.701,A -85,B 0,C 180,E1 26416.595,E2 26416.595} C_VEL
LIN {X 0,Y 697.797,Z 408.17,A -85,B 0,C 180,E1 26416.203,E2 26416.203} C_VEL
LIN {X 0,Y 702.472,Z 418.326,A -85,B 0,C 180,E1 26415.06,E2 26415.06} C_VEL
LIN {X 0,Y 711.32,Z 431.711,A -85,B 0,C 180,E1 26414.165,E2 26414.165} C_VEL
LIN {X 0,Y 712.351,Z 436.292,A -85,B 0,C 180,E1 26414.021,E2 26414.021} C_VEL
LIN {X 0,Y 710.474,Z 646.729,A -85,B 0,C 180,E1 26411.328,E2 26411.328} C_VEL
LIN {X 0,Y 708.642,Z 871.421,A -85,B 0,C 180,E1 26408.544,E2 26408.544} C_VEL
LIN {X 0,Y 708.213,Z 904.183,A -85,B 0,C 180,E1 26408.097,E2 26408.097} C_VEL
LIN {X 0,Y 707.571,Z 930.741,A -85,B 0,C 180,E1 26407.573,E2 26407.573} C_VEL
LIN {X 0,Y 706.887,Z 955.934,A -85,B 0,C 180,E1 26406.928,E2 26406.928} C_VEL
LIN {X 0,Y 705.972,Z 983.852,A -85,B 0,C 180,E1 26406.028,E2 26406.028} C_VEL
LIN {X 0,Y 705.103,Z 1006.563,A -85,B 0,C 180,E1 26405.152,E2 26405.152} C_VEL
LIN {X 0,Y 704.28,Z 1026.662,A -85,B 0,C 180,E1 26404.264,E2 26404.264} C_VEL
LIN {X 0,Y 703.426,Z 1046.465,A -85,B 0,C 180,E1 26403.278,E2 26403.278} C_VEL
LIN {X 0,Y 702.395,Z 1069.995,A -85,B 0,C 180,E1 26401.958,E2 26401.958} C_VEL
LIN {X 0,Y 701.391,Z 1092.593,A -85,B 0,C 180,E1 26400.499,E2 26400.499} C_VEL
LIN {X 0,Y 700.55,Z 1111.112,A -85,B 0,C 180,E1 26399.168,E2 26399.168} C_VEL
LIN {X 0,Y 699.716,Z 1130.481,A -85,B 0,C 180,E1 26397.628,E2 26397.628} C_VEL
LIN {X 0,Y 698.899,Z 1150.28,A -85,B 0,C 180,E1 26395.856,E2 26395.856} C_VEL
LIN {X 0,Y 698.266,Z 1166.245,A -85,B 0,C 180,E1 26394.267,E2 26394.267} C_VEL
LIN {X 0,Y 697.665,Z 1182.316,A -85,B 0,C 180,E1 26392.5,E2 26392.5} C_VEL
LIN {X 0,Y 697.116,Z 1199.177,A -85,B 0,C 180,E1 26390.4,E2 26390.4} C_VEL
LIN {X 0,Y 696.785,Z 1211.529,A -85,B 0,C 180,E1 26388.665,E2 26388.665} C_VEL
LIN {X 0,Y 696.5,Z 1223.029,A -85,B 0,C 180,E1 26386.859,E2 26386.859} C_VEL
LIN {X 0,Y 696.27,Z 1235.378,A -85,B 0,C 180,E1 26384.642,E2 26384.642} C_VEL
LIN {X 0,Y 696.099,Z 1245.235,A -85,B 0,C 180,E1 26382.529,E2 26382.529} C_VEL
LIN {X 0,Y 695.997,Z 1252.264,A -85,B 0,C 180,E1 26380.766,E2 26380.766} C_VEL
LIN {X 0,Y 695.917,Z 1257.906,A -85,B 0,C 180,E1 26379.096,E2 26379.096} C_VEL
LIN {X 0,Y 695.93,Z 1263.259,A -85,B 0,C 180,E1 26377.183,E2 26377.183} C_VEL
LIN {X 0,Y 695.918,Z 1267.845,A -85,B 0,C 180,E1 26374.948,E2 26374.948} C_VEL
LIN {X 0,Y 695.914,Z 1270.57,A -85,B 0,C 180,E1 26372.802,E2 26372.802} C_VEL
LIN {X 0,Y 695.877,Z 1271.724,A -85,B 0,C 180,E1 26370.99,E2 26370.99} C_VEL
LIN {X 0,Y 695.862,Z 1271.817,A -85,B 0,C 180,E1 26369.261,E2 26369.261} C_VEL
LIN {X 0,Y 695.903,Z 1270.918,A -85,B 0,C 180,E1 26367.532,E2 26367.532} C_VEL
LIN {X 0,Y 695.913,Z 1268.75,A -85,B 0,C 180,E1 26365.553,E2 26365.553} C_VEL
LIN {X 0,Y 695.923,Z 1264.655,A -85,B 0,C 180,E1 26363.32,E2 26363.32} C_VEL
LIN {X 0,Y 695.938,Z 1258.966,A -85,B 0,C 180,E1 26361.16,E2 26361.16} C_VEL
LIN {X 0,Y 695.991,Z 1252.897,A -85,B 0,C 180,E1 26359.317,E2 26359.317} C_VEL
LIN {X 0,Y 696.071,Z 1246.321,A -85,B 0,C 180,E1 26357.637,E2 26357.637} C_VEL
LIN {X 0,Y 696.184,Z 1238.299,A -85,B 0,C 180,E1 26355.871,E2 26355.871} C_VEL
LIN {X 0,Y 696.372,Z 1229,A -85,B 0,C 180,E1 26354.086,E2 26354.086} C_VEL
LIN {X 0,Y 696.661,Z 1215.639,A -85,B 0,C 180,E1 26351.857,E2 26351.857} C_VEL
LIN {X 0,Y 697.021,Z 1202.455,A -85,B 0,C 180,E1 26349.953,E2 26349.953} C_VEL
LIN {X 0,Y 697.437,Z 1189.547,A -85,B 0,C 180,E1 26348.282,E2 26348.282} C_VEL
LIN {X 0,Y 698.023,Z 1173.027,A -85,B 0,C 180,E1 26346.358,E2 26346.358} C_VEL
LIN {X 0,Y 698.708,Z 1154.812,A -85,B 0,C 180,E1 26344.489,E2 26344.489} C_VEL
LIN {X 0,Y 699.375,Z 1138.3,A -85,B 0,C 180,E1 26342.962,E2 26342.962} C_VEL
LIN {X 0,Y 700.278,Z 1117.729,A -85,B 0,C 180,E1 26341.241,E2 26341.241} C_VEL
LIN {X 0,Y 701.204,Z 1096.581,A -85,B 0,C 180,E1 26339.687,E2 26339.687} C_VEL
LIN {X 0,Y 702.053,Z 1077.821,A -85,B 0,C 180,E1 26338.443,E2 26338.443} C_VEL
LIN {X 0,Y 702.983,Z 1057.04,A -85,B 0,C 180,E1 26337.205,E2 26337.205} C_VEL
LIN {X 0,Y 704.095,Z 1030.679,A -85,B 0,C 180,E1 26335.835,E2 26335.835} C_VEL
LIN {X 0,Y 704.946,Z 1009.947,A -85,B 0,C 180,E1 26334.899,E2 26334.899} C_VEL
LIN {X 0,Y 705.719,Z 989.569,A -85,B 0,C 180,E1 26334.091,E2 26334.091} C_VEL
LIN {X 0,Y 706.48,Z 967.4,A -85,B 0,C 180,E1 26333.331,E2 26333.331} C_VEL
LIN {X 0,Y 707.308,Z 941.726,A -85,B 0,C 180,E1 26332.597,E2 26332.597} C_VEL
LIN {X 0,Y 707.987,Z 914.432,A -85,B 0,C 180,E1 26331.998,E2 26331.998} C_VEL
LIN {X 0,Y 708.444,Z 889.357,A -85,B 0,C 180,E1 26331.591,E2 26331.591} C_VEL
LIN {X 0,Y 710.337,Z 662.322,A -85,B 0,C 180,E1 26328.778,E2 26328.778} C_VEL
LIN {X 0,Y 712.13,Z 457.713,A -85,B 0,C 180,E1 26326.166,E2 26326.166} C_VEL
LIN {X 0,Y 712.191,Z 434.972,A -85,B 0,C 180,E1 26325.858,E2 26325.858} C_VEL
LIN {X 0,Y 710.838,Z 430.786,A -85,B 0,C 180,E1 26325.695,E2 26325.695} C_VEL
LIN {X 0,Y 702.021,Z 417.435,A -85,B 0,C 180,E1 26324.775,E2 26324.775} C_VEL
LIN {X 0,Y 697.704,Z 408.064,A -85,B 0,C 180,E1 26323.691,E2 26323.691} C_VEL
LIN {X 0,Y 696.353,Z 404.493,A -85,B 0,C 180,E1 26323.288,E2 26323.288} C_VEL
LIN {X 0,Y 696.383,Z 404.487,A -85,B 0,C 180,E1 26320.201,E2 26320.201} C_VEL
LIN {X 0,Y 696.335,Z 404.489,A -85,B 0,C 180,E1 26317.44,E2 26317.44} C_VEL
LIN {X 0,Y 696.387,Z 404.473,A -85,B 0,C 180,E1 26314.649,E2 26314.649} C_VEL
LIN {X 0,Y 696.347,Z 404.483,A -85,B 0,C 180,E1 26311.608,E2 26311.608} C_VEL
LIN {X 0,Y 696.333,Z 404.479,A -85,B 0,C 180,E1 26309.026,E2 26309.026} C_VEL
LIN {X 0,Y 696.4,Z 404.472,A -85,B 0,C 180,E1 26306.196,E2 26306.196} C_VEL
LIN {X 0,Y 696.336,Z 404.486,A -85,B 0,C 180,E1 26303.233,E2 26303.233} C_VEL
LIN {X 0,Y 696.33,Z 404.479,A -85,B 0,C 180,E1 26300.686,E2 26300.686} C_VEL
LIN {X 0,Y 696.407,Z 404.487,A -85,B 0,C 180,E1 26297.808,E2 26297.808} C_VEL
LIN {X 0,Y 696.327,Z 404.468,A -85,B 0,C 180,E1 26294.894,E2 26294.894} C_VEL
LIN {X 0,Y 696.329,Z 404.486,A -85,B 0,C 180,E1 26292.354,E2 26292.354} C_VEL
LIN {X 0,Y 696.404,Z 404.466,A -85,B 0,C 180,E1 26289.421,E2 26289.421} C_VEL
LIN {X 0,Y 696.327,Z 404.486,A -85,B 0,C 180,E1 26286.597,E2 26286.597} C_VEL
LIN {X 0,Y 696.322,Z 404.484,A -85,B 0,C 180,E1 26284.117,E2 26284.117} C_VEL
LIN {X 0,Y 696.404,Z 404.478,A -85,B 0,C 180,E1 26281.234,E2 26281.234} C_VEL
LIN {X 0,Y 696.326,Z 404.482,A -85,B 0,C 180,E1 26278.354,E2 26278.354} C_VEL
LIN {X 0,Y 696.316,Z 404.475,A -85,B 0,C 180,E1 26275.883,E2 26275.883} C_VEL
LIN {X 0,Y 696.376,Z 404.49,A -85,B 0,C 180,E1 26273.155,E2 26273.155} C_VEL
LIN {X 0,Y 696.33,Z 404.476,A -85,B 0,C 180,E1 26270.161,E2 26270.161} C_VEL
LIN {X 0,Y 696.312,Z 404.488,A -85,B 0,C 180,E1 26267.645,E2 26267.645} C_VEL
LIN {X 0,Y 696.341,Z 404.477,A -85,B 0,C 180,E1 26265.08,E2 26265.08} C_VEL
LIN {X 0,Y 696.332,Z 404.486,A -85,B 0,C 180,E1 26261.931,E2 26261.931} C_VEL
LIN {X 0,Y 696.307,Z 404.47,A -85,B 0,C 180,E1 26259.401,E2 26259.401} C_VEL
LIN {X 0,Y 696.326,Z 404.489,A -85,B 0,C 180,E1 26256.92,E2 26256.92} C_VEL
LIN {X 0,Y 696.348,Z 404.482,A -85,B 0,C 180,E1 26253.813,E2 26253.813} C_VEL
LIN {X 0,Y 696.307,Z 404.487,A -85,B 0,C 180,E1 26251.245,E2 26251.245} C_VEL
LIN {X 0,Y 696.307,Z 404.485,A -85,B 0,C 180,E1 26248.871,E2 26248.871} C_VEL
LIN {X 0,Y 696.386,Z 404.474,A -85,B 0,C 180,E1 26246.045,E2 26246.045} C_VEL
LIN {X 0,Y 696.31,Z 404.49,A -85,B 0,C 180,E1 26243.107,E2 26243.107} C_VEL
LIN {X 0,Y 696.3,Z 404.494,A -85,B 0,C 180,E1 26240.707,E2 26240.707} C_VEL
LIN {X 0,Y 696.312,Z 404.481,A -85,B 0,C 180,E1 26238.299,E2 26238.299} C_VEL
LIN {X 0,Y 696.379,Z 404.593,A -85,B 0,C 180,E1 26237.396,E2 26237.396} C_VEL
LIN {X 0,Y 697.772,Z 408.196,A -85,B 0,C 180,E1 26236.992,E2 26236.992} C_VEL
LIN {X 0,Y 703.989,Z 421.641,A -85,B 0,C 180,E1 26235.441,E2 26235.441} C_VEL
LIN {X 0,Y 707.092,Z 428.248,A -85,B 0,C 180,E1 26234.732,E2 26234.732} C_VEL
LIN {X 0,Y 708.576,Z 431.14,A -85,B 0,C 180,E1 26234.573,E2 26234.573} C_VEL
LIN {X 0,Y 712.312,Z 445.684,A -85,B 0,C 180,E1 26234.077,E2 26234.077} C_VEL
LIN {X 0,Y 710.571,Z 646.105,A -85,B 0,C 180,E1 26231.506,E2 26231.506} C_VEL
LIN {X 0,Y 708.721,Z 872.013,A -85,B 0,C 180,E1 26228.704,E2 26228.704} C_VEL
LIN {X 0,Y 708.26,Z 911.828,A -85,B 0,C 180,E1 26228.182,E2 26228.182} C_VEL
LIN {X 0,Y 707.616,Z 939.294,A -85,B 0,C 180,E1 26227.651,E2 26227.651} C_VEL
LIN {X 0,Y 706.928,Z 964.191,A -85,B 0,C 180,E1 26227.022,E2 26227.022} C_VEL
LIN {X 0,Y 706.055,Z 992.005,A -85,B 0,C 180,E1 26226.14,E2 26226.14} C_VEL
LIN {X 0,Y 705.146,Z 1015.587,A -85,B 0,C 180,E1 26225.238,E2 26225.238} C_VEL
LIN {X 0,Y 704.321,Z 1035.795,A -85,B 0,C 180,E1 26224.35,E2 26224.35} C_VEL
LIN {X 0,Y 703.47,Z 1055.611,A -85,B 0,C 180,E1 26223.367,E2 26223.367} C_VEL
LIN {X 0,Y 702.543,Z 1076.518,A -85,B 0,C 180,E1 26222.204,E2 26222.204} C_VEL
LIN {X 0,Y 701.453,Z 1101.303,A -85,B 0,C 180,E1 26220.633,E2 26220.633} C_VEL
LIN {X 0,Y 700.579,Z 1120.493,A -85,B 0,C 180,E1 26219.259,E2 26219.259} C_VEL
LIN {X 0,Y 699.801,Z 1138.71,A -85,B 0,C 180,E1 26217.817,E2 26217.817} C_VEL
LIN {X 0,Y 698.909,Z 1160.002,A -85,B 0,C 180,E1 26215.928,E2 26215.928} C_VEL
LIN {X 0,Y 698.283,Z 1175.867,A -85,B 0,C 180,E1 26214.352,E2 26214.352} C_VEL
LIN {X 0,Y 697.693,Z 1191.492,A -85,B 0,C 180,E1 26212.639,E2 26212.639} C_VEL
LIN {X 0,Y 697.136,Z 1208.667,A -85,B 0,C 180,E1 26210.513,E2 26210.513} C_VEL
LIN {X 0,Y 696.789,Z 1221.464,A -85,B 0,C 180,E1 26208.719,E2 26208.719} C_VEL
LIN {X 0,Y 696.511,Z 1232.808,A -85,B 0,C 180,E1 26206.94,E2 26206.94} C_VEL
LIN {X 0,Y 696.276,Z 1244.777,A -85,B 0,C 180,E1 26204.807,E2 26204.807} C_VEL
LIN {X 0,Y 696.106,Z 1255.089,A -85,B 0,C 180,E1 26202.608,E2 26202.608} C_VEL
LIN {X 0,Y 695.995,Z 1262.141,A -85,B 0,C 180,E1 26200.845,E2 26200.845} C_VEL
LIN {X 0,Y 695.917,Z 1267.803,A -85,B 0,C 180,E1 26199.174,E2 26199.174} C_VEL
LIN {X 0,Y 695.922,Z 1272.974,A -85,B 0,C 180,E1 26197.344,E2 26197.344} C_VEL
LIN {X 0,Y 695.915,Z 1277.638,A -85,B 0,C 180,E1 26195.108,E2 26195.108} C_VEL
LIN {X 0,Y 695.912,Z 1280.476,A -85,B 0,C 180,E1 26192.962,E2 26192.962} C_VEL
LIN {X 0,Y 695.877,Z 1281.715,A -85,B 0,C 180,E1 26191.068,E2 26191.068} C_VEL
LIN {X 0,Y 695.863,Z 1281.826,A -85,B 0,C 180,E1 26189.339,E2 26189.339} C_VEL
LIN {X 0,Y 695.905,Z 1280.944,A -85,B 0,C 180,E1 26187.61,E2 26187.61} C_VEL
LIN {X 0,Y 695.917,Z 1278.854,A -85,B 0,C 180,E1 26185.667,E2 26185.667} C_VEL
LIN {X 0,Y 695.927,Z 1274.73,A -85,B 0,C 180,E1 26183.398,E2 26183.398} C_VEL
LIN {X 0,Y 695.94,Z 1269.069,A -85,B 0,C 180,E1 26181.238,E2 26181.238} C_VEL
LIN {X 0,Y 695.997,Z 1263.041,A -85,B 0,C 180,E1 26179.402,E2 26179.402} C_VEL
LIN {X 0,Y 696.062,Z 1256.498,A -85,B 0,C 180,E1 26177.723,E2 26177.723} C_VEL
LIN {X 0,Y 696.176,Z 1248.469,A -85,B 0,C 180,E1 26175.951,E2 26175.951} C_VEL
LIN {X 0,Y 696.368,Z 1239.166,A -85,B 0,C 180,E1 26174.161,E2 26174.161} C_VEL
LIN {X 0,Y 696.654,Z 1225.882,A -85,B 0,C 180,E1 26171.938,E2 26171.938} C_VEL
LIN {X 0,Y 697.024,Z 1212.37,A -85,B 0,C 180,E1 26169.986,E2 26169.986} C_VEL
LIN {X 0,Y 697.451,Z 1199.157,A -85,B 0,C 180,E1 26168.279,E2 26168.279} C_VEL
LIN {X 0,Y 698.041,Z 1182.589,A -85,B 0,C 180,E1 26166.353,E2 26166.353} C_VEL
LIN {X 0,Y 698.731,Z 1164.297,A -85,B 0,C 180,E1 26164.485,E2 26164.485} C_VEL
LIN {X 0,Y 699.396,Z 1147.75,A -85,B 0,C 180,E1 26162.958,E2 26162.958} C_VEL
LIN {X 0,Y 700.303,Z 1127.075,A -85,B 0,C 180,E1 26161.237,E2 26161.237} C_VEL
LIN {X 0,Y 701.204,Z 1106.534,A -85,B 0,C 180,E1 26159.729,E2 26159.729} C_VEL
LIN {X 0,Y 702.053,Z 1087.776,A -85,B 0,C 180,E1 26158.486,E2 26158.486} C_VEL
LIN {X 0,Y 702.957,Z 1067.567,A -85,B 0,C 180,E1 26157.28,E2 26157.28} C_VEL
LIN {X 0,Y 704.057,Z 1041.545,A -85,B 0,C 180,E1 26155.92,E2 26155.92} C_VEL
LIN {X 0,Y 704.97,Z 1019.463,A -85,B 0,C 180,E1 26154.924,E2 26154.924} C_VEL
LIN {X 0,Y 705.778,Z 998.281,A -85,B 0,C 180,E1 26154.089,E2 26154.089} C_VEL
LIN {X 0,Y 706.615,Z 973.693,A -85,B 0,C 180,E1 26153.257,E2 26153.257} C_VEL
LIN {X 0,Y 707.453,Z 946.217,A -85,B 0,C 180,E1 26152.509,E2 26152.509} C_VEL
LIN {X 0,Y 708.046,Z 921.044,A -85,B 0,C 180,E1 26151.98,E2 26151.98} C_VEL
LIN {X 0,Y 708.522,Z 894.386,A -85,B 0,C 180,E1 26151.57,E2 26151.57} C_VEL
LIN {X 0,Y 710.376,Z 667.811,A -85,B 0,C 180,E1 26148.766,E2 26148.766} C_VEL
LIN {X 0,Y 712.085,Z 470.303,A -85,B 0,C 180,E1 26146.243,E2 26146.243} C_VEL
LIN {X 0,Y 712.168,Z 444.495,A -85,B 0,C 180,E1 26145.895,E2 26145.895} C_VEL
LIN {X 0,Y 707.951,Z 429.62,A -85,B 0,C 180,E1 26145.356,E2 26145.356} C_VEL
LIN {X 0,Y 706.433,Z 427.115,A -85,B 0,C 180,E1 26145.164,E2 26145.164} C_VEL
LIN {X 0,Y 699.845,Z 412.553,A -85,B 0,C 180,E1 26143.523,E2 26143.523} C_VEL
LIN {X 0,Y 696.476,Z 405.176,A -85,B 0,C 180,E1 26142.658,E2 26142.658} C_VEL
LIN {X 0,Y 696.378,Z 404.492,A -85,B 0,C 180,E1 26142.554,E2 26142.554} C_VEL
LIN {X 0,Y 696.308,Z 404.495,A -85,B 0,C 180,E1 26139.612,E2 26139.612} C_VEL
LIN {X 0,Y 696.306,Z 404.483,A -85,B 0,C 180,E1 26137.157,E2 26137.157} C_VEL
LIN {X 0,Y 696.373,Z 404.476,A -85,B 0,C 180,E1 26134.453,E2 26134.453} C_VEL
LIN {X 0,Y 696.326,Z 404.487,A -85,B 0,C 180,E1 26131.466,E2 26131.466} C_VEL
LIN {X 0,Y 696.317,Z 404.481,A -85,B 0,C 180,E1 26129.014,E2 26129.014} C_VEL
LIN {X 0,Y 696.372,Z 404.481,A -85,B 0,C 180,E1 26126.339,E2 26126.339} C_VEL
LIN {X 0,Y 696.344,Z 404.486,A -85,B 0,C 180,E1 26123.348,E2 26123.348} C_VEL
LIN {X 0,Y 696.331,Z 404.479,A -85,B 0,C 180,E1 26120.774,E2 26120.774} C_VEL
LIN {X 0,Y 696.402,Z 404.487,A -85,B 0,C 180,E1 26117.981,E2 26117.981} C_VEL
LIN {X 0,Y 696.344,Z 404.467,A -85,B 0,C 180,E1 26114.979,E2 26114.979} C_VEL
LIN {X 0,Y 696.361,Z 404.486,A -85,B 0,C 180,E1 26112.27,E2 26112.27} C_VEL
LIN {X 0,Y 696.384,Z 404.464,A -85,B 0,C 180,E1 26109.171,E2 26109.171} C_VEL
LIN {X 0,Y 696.354,Z 404.485,A -85,B 0,C 180,E1 26106.348,E2 26106.348} C_VEL
LIN {X 0,Y 696.397,Z 404.466,A -85,B 0,C 180,E1 26103.457,E2 26103.457} C_VEL
LIN {X 0,Y 696.361,Z 404.482,A -85,B 0,C 180,E1 26100.494,E2 26100.494} C_VEL
LIN {X 0,Y 696.398,Z 404.469,A -85,B 0,C 180,E1 26097.614,E2 26097.614} C_VEL
LIN {X 0,Y 696.38,Z 404.479,A -85,B 0,C 180,E1 26094.562,E2 26094.562} C_VEL
LIN {X 0,Y 696.399,Z 404.471,A -85,B 0,C 180,E1 26091.579,E2 26091.579} C_VEL
LIN {X 0,Y 696.394,Z 404.478,A -85,B 0,C 180,E1 26088.488,E2 26088.488} C_VEL
LIN {X 0,Y 696.399,Z 404.47,A -85,B 0,C 180,E1 26085.403,E2 26085.403} C_VEL
LIN {X 0,Y 696.396,Z 404.479,A -85,B 0,C 180,E1 26082.278,E2 26082.278} C_VEL
LIN {X 0,Y 696.394,Z 404.472,A -85,B 0,C 180,E1 26079.181,E2 26079.181} C_VEL
LIN {X 0,Y 696.399,Z 404.477,A -85,B 0,C 180,E1 26076.115,E2 26076.115} C_VEL
LIN {X 0,Y 696.396,Z 404.473,A -85,B 0,C 180,E1 26075.204,E2 26075.204} C_VEL
LIN {X 0,Y 695.388,Z 404.592,A -85,B 0,C 180,E1 26074.57,E2 26074.57} C_VEL
LIN {X 0,Y 688.96,Z 405.411,A -85,B 0,C 180,E1 26072.795,E2 26072.795} C_VEL
LIN {X 0,Y 688.447,Z 405.47,A -85,B 0,C 180,E1 26072.333,E2 26072.333} C_VEL
LIN {X 0,Y 688.46,Z 405.459,A -85,B 0,C 180,E1 26069.254,E2 26069.254} C_VEL
LIN {X 0,Y 688.431,Z 405.462,A -85,B 0,C 180,E1 26066.301,E2 26066.301} C_VEL
LIN {X 0,Y 688.459,Z 405.476,A -85,B 0,C 180,E1 26063.293,E2 26063.293} C_VEL
LIN {X 0,Y 688.424,Z 405.479,A -85,B 0,C 180,E1 26060.385,E2 26060.385} C_VEL
LIN {X 0,Y 688.462,Z 405.466,A -85,B 0,C 180,E1 26057.519,E2 26057.519} C_VEL
LIN {X 0,Y 688.474,Z 405.566,A -85,B 0,C 180,E1 26057.229,E2 26057.229} C_VEL
LIN {X 0,Y 689.817,Z 409.046,A -85,B 0,C 180,E1 26056.83,E2 26056.83} C_VEL
LIN {X 0,Y 694.228,Z 418.34,A -85,B 0,C 180,E1 26055.747,E2 26055.747} C_VEL
LIN {X 0,Y 706.234,Z 436.529,A -85,B 0,C 180,E1 26054.5,E2 26054.5} C_VEL
LIN {X 0,Y 706.561,Z 439.115,A -85,B 0,C 180,E1 26054.438,E2 26054.438} C_VEL
LIN {X 0,Y 704.444,Z 648.561,A -85,B 0,C 180,E1 26051.737,E2 26051.737} C_VEL
LIN {X 0,Y 702.368,Z 873.125,A -85,B 0,C 180,E1 26048.932,E2 26048.932} C_VEL
LIN {X 0,Y 701.869,Z 905.423,A -85,B 0,C 180,E1 26048.481,E2 26048.481} C_VEL
LIN {X 0,Y 701.172,Z 931.125,A -85,B 0,C 180,E1 26047.967,E2 26047.967} C_VEL
LIN {X 0,Y 700.4,Z 956.207,A -85,B 0,C 180,E1 26047.32,E2 26047.32} C_VEL
LIN {X 0,Y 699.402,Z 983.289,A -85,B 0,C 180,E1 26046.443,E2 26046.443} C_VEL
LIN {X 0,Y 698.433,Z 1005.892,A -85,B 0,C 180,E1 26045.569,E2 26045.569} C_VEL
LIN {X 0,Y 697.485,Z 1026.475,A -85,B 0,C 180,E1 26044.655,E2 26044.655} C_VEL
LIN {X 0,Y 696.556,Z 1045.59,A -85,B 0,C 180,E1 26043.699,E2 26043.699} C_VEL
LIN {X 0,Y 695.562,Z 1065.684,A -85,B 0,C 180,E1 26042.573,E2 26042.573} C_VEL
LIN {X 0,Y 694.274,Z 1090.596,A -85,B 0,C 180,E1 26040.99,E2 26040.99} C_VEL
LIN {X 0,Y 693.283,Z 1110.169,A -85,B 0,C 180,E1 26039.578,E2 26039.578} C_VEL
LIN {X 0,Y 692.394,Z 1128.454,A -85,B 0,C 180,E1 26038.117,E2 26038.117} C_VEL
LIN {X 0,Y 691.341,Z 1150.116,A -85,B 0,C 180,E1 26036.177,E2 26036.177} C_VEL
LIN {X 0,Y 690.629,Z 1166.252,A -85,B 0,C 180,E1 26034.553,E2 26034.553} C_VEL
LIN {X 0,Y 689.912,Z 1183.09,A -85,B 0,C 180,E1 26032.677,E2 26032.677} C_VEL
LIN {X 0,Y 689.312,Z 1199.183,A -85,B 0,C 180,E1 26030.641,E2 26030.641} C_VEL
LIN {X 0,Y 688.92,Z 1211.706,A -85,B 0,C 180,E1 26028.86,E2 26028.86} C_VEL
LIN {X 0,Y 688.599,Z 1223.034,A -85,B 0,C 180,E1 26027.058,E2 26027.058} C_VEL
LIN {X 0,Y 688.32,Z 1235.382,A -85,B 0,C 180,E1 26024.815,E2 26024.815} C_VEL
LIN {X 0,Y 688.136,Z 1245.238,A -85,B 0,C 180,E1 26022.676,E2 26022.676} C_VEL
LIN {X 0,Y 688.013,Z 1252.267,A -85,B 0,C 180,E1 26020.892,E2 26020.892} C_VEL
LIN {X 0,Y 687.924,Z 1257.908,A -85,B 0,C 180,E1 26019.202,E2 26019.202} C_VEL
LIN {X 0,Y 687.92,Z 1263.054,A -85,B 0,C 180,E1 26017.351,E2 26017.351} C_VEL
LIN {X 0,Y 687.917,Z 1267.698,A -85,B 0,C 180,E1 26015.089,E2 26015.089} C_VEL
LIN {X 0,Y 687.912,Z 1270.503,A -85,B 0,C 180,E1 26012.918,E2 26012.918} C_VEL
LIN {X 0,Y 687.878,Z 1271.724,A -85,B 0,C 180,E1 26011.002,E2 26011.002} C_VEL
LIN {X 0,Y 687.863,Z 1271.817,A -85,B 0,C 180,E1 26009.253,E2 26009.253} C_VEL
LIN {X 0,Y 687.903,Z 1270.917,A -85,B 0,C 180,E1 26007.503,E2 26007.503} C_VEL
LIN {X 0,Y 687.914,Z 1268.873,A -85,B 0,C 180,E1 26005.584,E2 26005.584} C_VEL
LIN {X 0,Y 687.925,Z 1264.833,A -85,B 0,C 180,E1 26003.325,E2 26003.325} C_VEL
LIN {X 0,Y 687.943,Z 1259.221,A -85,B 0,C 180,E1 26001.14,E2 26001.14} C_VEL
LIN {X 0,Y 688.002,Z 1253.109,A -85,B 0,C 180,E1 25999.251,E2 25999.251} C_VEL
LIN {X 0,Y 688.107,Z 1246.352,A -85,B 0,C 180,E1 25997.499,E2 25997.499} C_VEL
LIN {X 0,Y 688.247,Z 1238.29,A -85,B 0,C 180,E1 25995.703,E2 25995.703} C_VEL
LIN {X 0,Y 688.446,Z 1228.533,A -85,B 0,C 180,E1 25993.811,E2 25993.811} C_VEL
LIN {X 0,Y 688.816,Z 1215.06,A -85,B 0,C 180,E1 25991.555,E2 25991.555} C_VEL
LIN {X 0,Y 689.195,Z 1202.453,A -85,B 0,C 180,E1 25989.715,E2 25989.715} C_VEL
LIN {X 0,Y 689.699,Z 1188.935,A -85,B 0,C 180,E1 25987.949,E2 25987.949} C_VEL
LIN {X 0,Y 690.404,Z 1171.38,A -85,B 0,C 180,E1 25985.899,E2 25985.899} C_VEL
LIN {X 0,Y 691.205,Z 1153.445,A -85,B 0,C 180,E1 25984.057,E2 25984.057} C_VEL
LIN {X 0,Y 691.977,Z 1136.267,A -85,B 0,C 180,E1 25982.463,E2 25982.463} C_VEL
LIN {X 0,Y 693.105,Z 1113.895,A -85,B 0,C 180,E1 25980.616,E2 25980.616} C_VEL
LIN {X 0,Y 694.057,Z 1095.249,A -85,B 0,C 180,E1 25979.245,E2 25979.245} C_VEL
LIN {X 0,Y 695.012,Z 1076.35,A -85,B 0,C 180,E1 25977.989,E2 25977.989} C_VEL
LIN {X 0,Y 696.242,Z 1052.058,A -85,B 0,C 180,E1 25976.553,E2 25976.553} C_VEL
LIN {X 0,Y 697.372,Z 1028.78,A -85,B 0,C 180,E1 25975.364,E2 25975.364} C_VEL
LIN {X 0,Y 698.298,Z 1008.706,A -85,B 0,C 180,E1 25974.459,E2 25974.459} C_VEL
LIN {X 0,Y 699.175,Z 988.149,A -85,B 0,C 180,E1 25973.646,E2 25973.646} C_VEL
LIN {X 0,Y 700.076,Z 964.417,A -85,B 0,C 180,E1 25972.837,E2 25972.837} C_VEL
LIN {X 0,Y 701.018,Z 937.171,A -85,B 0,C 180,E1 25972.084,E2 25972.084} C_VEL
LIN {X 0,Y 701.691,Z 911.936,A -85,B 0,C 180,E1 25971.546,E2 25971.546} C_VEL
LIN {X 0,Y 702.222,Z 886.076,A -85,B 0,C 180,E1 25971.14,E2 25971.14} C_VEL
LIN {X 0,Y 704.332,Z 659.934,A -85,B 0,C 180,E1 25968.317,E2 25968.317} C_VEL
LIN {X 0,Y 706.381,Z 454.593,A -85,B 0,C 180,E1 25965.674,E2 25965.674} C_VEL
LIN {X 0,Y 706.401,Z 437.209,A -85,B 0,C 180,E1 25965.433,E2 25965.433} C_VEL
LIN {X 0,Y 705.393,Z 434.952,A -85,B 0,C 180,E1 25965.321,E2 25965.321} C_VEL
LIN {X 0,Y 693.868,Z 417.636,A -85,B 0,C 180,E1 25964.109,E2 25964.109} C_VEL
LIN {X 0,Y 688.534,Z 405.92,A -85,B 0,C 180,E1 25962.715,E2 25962.715} C_VEL
LIN {X 0,Y 688.467,Z 405.471,A -85,B 0,C 180,E1 25962.657,E2 25962.657} C_VEL
LIN {X 0,Y 688.402,Z 405.479,A -85,B 0,C 180,E1 25959.724,E2 25959.724} C_VEL
LIN {X 0,Y 688.412,Z 405.477,A -85,B 0,C 180,E1 25957.069,E2 25957.069} C_VEL
LIN {X 0,Y 688.44,Z 405.461,A -85,B 0,C 180,E1 25953.98,E2 25953.98} C_VEL
LIN {X 0,Y 688.394,Z 405.474,A -85,B 0,C 180,E1 25951.235,E2 25951.235} C_VEL
LIN {X 0,Y 688.434,Z 405.47,A -85,B 0,C 180,E1 25948.523,E2 25948.523} C_VEL
LIN {X 0,Y 688.404,Z 405.457,A -85,B 0,C 180,E1 25945.398,E2 25945.398} C_VEL
LIN {X 0,Y 688.39,Z 405.477,A -85,B 0,C 180,E1 25942.819,E2 25942.819} C_VEL
LIN {X 0,Y 688.463,Z 405.457,A -85,B 0,C 180,E1 25939.956,E2 25939.956} C_VEL
LIN {X 0,Y 688.393,Z 405.474,A -85,B 0,C 180,E1 25936.975,E2 25936.975} C_VEL
LIN {X 0,Y 688.386,Z 405.457,A -85,B 0,C 180,E1 25934.468,E2 25934.468} C_VEL
LIN {X 0,Y 688.466,Z 405.473,A -85,B 0,C 180,E1 25931.562,E2 25931.562} C_VEL
LIN {X 0,Y 688.388,Z 405.457,A -85,B 0,C 180,E1 25928.688,E2 25928.688} C_VEL
LIN {X 0,Y 688.386,Z 405.476,A -85,B 0,C 180,E1 25926.17,E2 25926.17} C_VEL
LIN {X 0,Y 688.464,Z 405.454,A -85,B 0,C 180,E1 25923.247,E2 25923.247} C_VEL
LIN {X 0,Y 688.386,Z 405.475,A -85,B 0,C 180,E1 25920.333,E2 25920.333} C_VEL
LIN {X 0,Y 688.383,Z 405.472,A -85,B 0,C 180,E1 25917.836,E2 25917.836} C_VEL
LIN {X 0,Y 688.464,Z 405.47,A -85,B 0,C 180,E1 25914.917,E2 25914.917} C_VEL
LIN {X 0,Y 688.38,Z 405.47,A -85,B 0,C 180,E1 25912.068,E2 25912.068} C_VEL
LIN {X 0,Y 688.376,Z 405.466,A -85,B 0,C 180,E1 25909.624,E2 25909.624} C_VEL
LIN {X 0,Y 688.452,Z 405.472,A -85,B 0,C 180,E1 25906.819,E2 25906.819} C_VEL
LIN {X 0,Y 688.384,Z 405.469,A -85,B 0,C 180,E1 25903.893,E2 25903.893} C_VEL
LIN {X 0,Y 688.371,Z 405.476,A -85,B 0,C 180,E1 25901.451,E2 25901.451} C_VEL
LIN {X 0,Y 688.395,Z 405.458,A -85,B 0,C 180,E1 25898.886,E2 25898.886} C_VEL
LIN {X 0,Y 688.392,Z 405.469,A -85,B 0,C 180,E1 25895.729,E2 25895.729} C_VEL
LIN {X 0,Y 688.367,Z 405.475,A -85,B 0,C 180,E1 25893.237,E2 25893.237} C_VEL
LIN {X 0,Y 688.377,Z 405.477,A -85,B 0,C 180,E1 25890.787,E2 25890.787} C_VEL
LIN {X 0,Y 688.445,Z 405.477,A -85,B 0,C 180,E1 25887.85,E2 25887.85} C_VEL
LIN {X 0,Y 688.367,Z 405.476,A -85,B 0,C 180,E1 25885.089,E2 25885.089} C_VEL
LIN {X 0,Y 688.364,Z 405.48,A -85,B 0,C 180,E1 25882.719,E2 25882.719} C_VEL
LIN {X 0,Y 688.409,Z 405.478,A -85,B 0,C 180,E1 25880.059,E2 25880.059} C_VEL
LIN {X 0,Y 688.424,Z 405.647,A -85,B 0,C 180,E1 25878.036,E2 25878.036} C_VEL
LIN {X 0,Y 689.876,Z 409.124,A -85,B 0,C 180,E1 25877.626,E2 25877.626} C_VEL
LIN {X 0,Y 697.734,Z 426.116,A -85,B 0,C 180,E1 25875.626,E2 25875.626} C_VEL
LIN {X 0,Y 698.863,Z 428.465,A -85,B 0,C 180,E1 25875.401,E2 25875.401} C_VEL
LIN {X 0,Y 703.335,Z 435.293,A -85,B 0,C 180,E1 25874.936,E2 25874.936} C_VEL
LIN {X 0,Y 706.53,Z 448.021,A -85,B 0,C 180,E1 25874.5,E2 25874.5} C_VEL
LIN {X 0,Y 704.547,Z 648.522,A -85,B 0,C 180,E1 25871.909,E2 25871.909} C_VEL
LIN {X 0,Y 702.455,Z 873.83,A -85,B 0,C 180,E1 25869.091,E2 25869.091} C_VEL
LIN {X 0,Y 701.943,Z 912.274,A -85,B 0,C 180,E1 25868.581,E2 25868.581} C_VEL
LIN {X 0,Y 701.225,Z 939.567,A -85,B 0,C 180,E1 25868.048,E2 25868.048} C_VEL
LIN {X 0,Y 700.449,Z 964.283,A -85,B 0,C 180,E1 25867.419,E2 25867.419} C_VEL
LIN {X 0,Y 699.48,Z 991.689,A -85,B 0,C 180,E1 25866.547,E2 25866.547} C_VEL
LIN {X 0,Y 698.453,Z 1015.45,A -85,B 0,C 180,E1 25865.632,E2 25865.632} C_VEL
LIN {X 0,Y 697.52,Z 1035.798,A -85,B 0,C 180,E1 25864.732,E2 25864.732} C_VEL
LIN {X 0,Y 696.558,Z 1055.614,A -85,B 0,C 180,E1 25863.742,E2 25863.742} C_VEL
LIN {X 0,Y 695.551,Z 1075.913,A -85,B 0,C 180,E1 25862.605,E2 25862.605} C_VEL
LIN {X 0,Y 694.272,Z 1100.708,A -85,B 0,C 180,E1 25861.027,E2 25861.027} C_VEL
LIN {X 0,Y 693.296,Z 1119.889,A -85,B 0,C 180,E1 25859.645,E2 25859.645} C_VEL
LIN {X 0,Y 692.447,Z 1137.322,A -85,B 0,C 180,E1 25858.256,E2 25858.256} C_VEL
LIN {X 0,Y 691.466,Z 1157.482,A -85,B 0,C 180,E1 25856.478,E2 25856.478} C_VEL
LIN {X 0,Y 690.675,Z 1175.015,A -85,B 0,C 180,E1 25854.729,E2 25854.729} C_VEL
LIN {X 0,Y 690.019,Z 1190.436,A -85,B 0,C 180,E1 25853.029,E2 25853.029} C_VEL
LIN {X 0,Y 689.382,Z 1207.612,A -85,B 0,C 180,E1 25850.9,E2 25850.9} C_VEL
LIN {X 0,Y 688.936,Z 1221.283,A -85,B 0,C 180,E1 25848.968,E2 25848.968} C_VEL
LIN {X 0,Y 688.605,Z 1232.81,A -85,B 0,C 180,E1 25847.14,E2 25847.14} C_VEL
LIN {X 0,Y 688.323,Z 1244.786,A -85,B 0,C 180,E1 25844.98,E2 25844.98} C_VEL
LIN {X 0,Y 688.14,Z 1255.09,A -85,B 0,C 180,E1 25842.757,E2 25842.757} C_VEL
LIN {X 0,Y 688.013,Z 1262.142,A -85,B 0,C 180,E1 25840.972,E2 25840.972} C_VEL
LIN {X 0,Y 687.924,Z 1267.821,A -85,B 0,C 180,E1 25839.276,E2 25839.276} C_VEL
LIN {X 0,Y 687.918,Z 1272.971,A -85,B 0,C 180,E1 25837.43,E2 25837.43} C_VEL
LIN {X 0,Y 687.914,Z 1277.49,A -85,B 0,C 180,E1 25835.251,E2 25835.251} C_VEL
LIN {X 0,Y 687.91,Z 1280.423,A -85,B 0,C 180,E1 25833.062,E2 25833.062} C_VEL
LIN {X 0,Y 687.879,Z 1281.715,A -85,B 0,C 180,E1 25831.08,E2 25831.08} C_VEL
LIN {X 0,Y 687.863,Z 1281.826,A -85,B 0,C 180,E1 25829.331,E2 25829.331} C_VEL
LIN {X 0,Y 687.905,Z 1280.944,A -85,B 0,C 180,E1 25827.582,E2 25827.582} C_VEL
LIN {X 0,Y 687.916,Z 1278.892,A -85,B 0,C 180,E1 25825.643,E2 25825.643} C_VEL
LIN {X 0,Y 687.927,Z 1274.73,A -85,B 0,C 180,E1 25823.321,E2 25823.321} C_VEL
LIN {X 0,Y 687.938,Z 1269.069,A -85,B 0,C 180,E1 25821.135,E2 25821.135} C_VEL
LIN {X 0,Y 688.006,Z 1263.042,A -85,B 0,C 180,E1 25819.277,E2 25819.277} C_VEL
LIN {X 0,Y 688.111,Z 1256.142,A -85,B 0,C 180,E1 25817.494,E2 25817.494} C_VEL
LIN {X 0,Y 688.254,Z 1248.06,A -85,B 0,C 180,E1 25815.7,E2 25815.7} C_VEL
LIN {X 0,Y 688.461,Z 1237.801,A -85,B 0,C 180,E1 25813.72,E2 25813.72} C_VEL
LIN {X 0,Y 688.86,Z 1223.83,A -85,B 0,C 180,E1 25811.414,E2 25811.414} C_VEL
LIN {X 0,Y 689.236,Z 1211.145,A -85,B 0,C 180,E1 25809.582,E2 25809.582} C_VEL
LIN {X 0,Y 689.773,Z 1197.116,A -85,B 0,C 180,E1 25807.767,E2 25807.767} C_VEL
LIN {X 0,Y 690.54,Z 1178.271,A -85,B 0,C 180,E1 25805.614,E2 25805.614} C_VEL
LIN {X 0,Y 691.247,Z 1162.434,A -85,B 0,C 180,E1 25804.004,E2 25804.004} C_VEL
LIN {X 0,Y 692.122,Z 1143.688,A -85,B 0,C 180,E1 25802.277,E2 25802.277} C_VEL
LIN {X 0,Y 693.134,Z 1123.247,A -85,B 0,C 180,E1 25800.612,E2 25800.612} C_VEL
LIN {X 0,Y 694.09,Z 1104.549,A -85,B 0,C 180,E1 25799.241,E2 25799.241} C_VEL
LIN {X 0,Y 695.115,Z 1084.112,A -85,B 0,C 180,E1 25797.892,E2 25797.892} C_VEL
LIN {X 0,Y 696.385,Z 1059.071,A -85,B 0,C 180,E1 25796.44,E2 25796.44} C_VEL
LIN {X 0,Y 697.397,Z 1038.248,A -85,B 0,C 180,E1 25795.384,E2 25795.384} C_VEL
LIN {X 0,Y 698.298,Z 1018.699,A -85,B 0,C 180,E1 25794.504,E2 25794.504} C_VEL
LIN {X 0,Y 699.169,Z 998.278,A -85,B 0,C 180,E1 25793.695,E2 25793.695} C_VEL
LIN {X 0,Y 700.075,Z 974.43,A -85,B 0,C 180,E1 25792.883,E2 25792.883} C_VEL
LIN {X 0,Y 701.018,Z 947.205,A -85,B 0,C 180,E1 25792.13,E2 25792.13} C_VEL
LIN {X 0,Y 701.691,Z 921.977,A -85,B 0,C 180,E1 25791.592,E2 25791.592} C_VEL
LIN {X 0,Y 702.22,Z 896.232,A -85,B 0,C 180,E1 25791.187,E2 25791.187} C_VEL
LIN {X 0,Y 704.338,Z 669.321,A -85,B 0,C 180,E1 25788.355,E2 25788.355} C_VEL
LIN {X 0,Y 706.287,Z 471.324,A -85,B 0,C 180,E1 25785.805,E2 25785.805} C_VEL
LIN {X 0,Y 706.386,Z 446.738,A -85,B 0,C 180,E1 25785.47,E2 25785.47} C_VEL
LIN {X 0,Y 702.929,Z 434.369,A -85,B 0,C 180,E1 25785.018,E2 25785.018} C_VEL
LIN {X 0,Y 698.229,Z 427.342,A -85,B 0,C 180,E1 25784.507,E2 25784.507} C_VEL
LIN {X 0,Y 691.813,Z 413.338,A -85,B 0,C 180,E1 25782.88,E2 25782.88} C_VEL
LIN {X 0,Y 689.56,Z 408.67,A -85,B 0,C 180,E1 25782.309,E2 25782.309} C_VEL
LIN {X 0,Y 688.384,Z 405.471,A -85,B 0,C 180,E1 25781.925,E2 25781.925} C_VEL
LIN {X 0,Y 688.362,Z 405.485,A -85,B 0,C 180,E1 25779.397,E2 25779.397} C_VEL
LIN {X 0,Y 688.386,Z 405.472,A -85,B 0,C 180,E1 25776.862,E2 25776.862} C_VEL
LIN {X 0,Y 688.396,Z 405.468,A -85,B 0,C 180,E1 25773.701,E2 25773.701} C_VEL
LIN {X 0,Y 688.376,Z 405.477,A -85,B 0,C 180,E1 25771.138,E2 25771.138} C_VEL
LIN {X 0,Y 688.41,Z 405.471,A -85,B 0,C 180,E1 25768.546,E2 25768.546} C_VEL
LIN {X 0,Y 688.407,Z 405.458,A -85,B 0,C 180,E1 25765.463,E2 25765.463} C_VEL
LIN {X 0,Y 688.388,Z 405.477,A -85,B 0,C 180,E1 25762.909,E2 25762.909} C_VEL
LIN {X 0,Y 688.447,Z 405.459,A -85,B 0,C 180,E1 25760.134,E2 25760.134} C_VEL
LIN {X 0,Y 688.41,Z 405.473,A -85,B 0,C 180,E1 25757.115,E2 25757.115} C_VEL
LIN {X 0,Y 688.405,Z 405.457,A -85,B 0,C 180,E1 25754.467,E2 25754.467} C_VEL
LIN {X 0,Y 688.463,Z 405.469,A -85,B 0,C 180,E1 25751.477,E2 25751.477} C_VEL
LIN {X 0,Y 688.408,Z 405.455,A -85,B 0,C 180,E1 25748.604,E2 25748.604} C_VEL
LIN {X 0,Y 688.464,Z 405.475,A -85,B 0,C 180,E1 25745.751,E2 25745.751} C_VEL
LIN {X 0,Y 688.422,Z 405.453,A -85,B 0,C 180,E1 25742.664,E2 25742.664} C_VEL
LIN {X 0,Y 688.458,Z 405.478,A -85,B 0,C 180,E1 25739.75,E2 25739.75} C_VEL
LIN {X 0,Y 688.442,Z 405.451,A -85,B 0,C 180,E1 25736.669,E2 25736.669} C_VEL
LIN {X 0,Y 688.456,Z 405.478,A -85,B 0,C 180,E1 25733.663,E2 25733.663} C_VEL
LIN {X 0,Y 688.452,Z 405.451,A -85,B 0,C 180,E1 25730.554,E2 25730.554} C_VEL
LIN {X 0,Y 688.46,Z 405.476,A -85,B 0,C 180,E1 25727.502,E2 25727.502} C_VEL
LIN {X 0,Y 688.454,Z 405.455,A -85,B 0,C 180,E1 25724.327,E2 25724.327} C_VEL
LIN {X 0,Y 688.459,Z 405.468,A -85,B 0,C 180,E1 25721.251,E2 25721.251} C_VEL
LIN {X 0,Y 688.458,Z 405.463,A -85,B 0,C 180,E1 25718.134,E2 25718.134} C_VEL
LIN {X 0,Y 688.452,Z 405.458,A -85,B 0,C 180,E1 25715.09,E2 25715.09} C_VEL
LIN {X 0,Y 688.447,Z 405.47,A -85,B 0,C 180,E1 25712.333,E2 25712.333} C_VEL
LIN {X 0,Y 687.477,Z 405.596,A -85,B 0,C 180,E1 25711.692,E2 25711.692} C_VEL
LIN {X 0,Y 681.038,Z 406.378,A -85,B 0,C 180,E1 25709.896,E2 25709.896} C_VEL
LIN {X 0,Y 680.514,Z 406.444,A -85,B 0,C 180,E1 25709.429,E2 25709.429} C_VEL
LIN {X 0,Y 680.49,Z 406.452,A -85,B 0,C 180,E1 25706.462,E2 25706.462} C_VEL
LIN {X 0,Y 680.519,Z 406.464,A -85,B 0,C 180,E1 25703.482,E2 25703.482} C_VEL
LIN {X 0,Y 680.487,Z 406.469,A -85,B 0,C 180,E1 25700.482,E2 25700.482} C_VEL
LIN {X 0,Y 680.515,Z 406.592,A -85,B 0,C 180,E1 25697.875,E2 25697.875} C_VEL
LIN {X 0,Y 681.878,Z 410.011,A -85,B 0,C 180,E1 25697.468,E2 25697.468} C_VEL
LIN {X 0,Y 685.828,Z 418.363,A -85,B 0,C 180,E1 25696.473,E2 25696.473} C_VEL
LIN {X 0,Y 700.827,Z 440.499,A -85,B 0,C 180,E1 25694.88,E2 25694.88} C_VEL
LIN {X 0,Y 698.461,Z 649.59,A -85,B 0,C 180,E1 25692.163,E2 25692.163} C_VEL
LIN {X 0,Y 696.136,Z 873.813,A -85,B 0,C 180,E1 25689.339,E2 25689.339} C_VEL
LIN {X 0,Y 695.571,Z 906.147,A -85,B 0,C 180,E1 25688.881,E2 25688.881} C_VEL
LIN {X 0,Y 694.81,Z 931.47,A -85,B 0,C 180,E1 25688.369,E2 25688.369} C_VEL
LIN {X 0,Y 693.938,Z 956.693,A -85,B 0,C 180,E1 25687.713,E2 25687.713} C_VEL
LIN {X 0,Y 692.777,Z 984.586,A -85,B 0,C 180,E1 25686.797,E2 25686.797} C_VEL
LIN {X 0,Y 691.756,Z 1006.07,A -85,B 0,C 180,E1 25685.958,E2 25685.958} C_VEL
LIN {X 0,Y 690.747,Z 1025.797,A -85,B 0,C 180,E1 25685.078,E2 25685.078} C_VEL
LIN {X 0,Y 689.675,Z 1045.605,A -85,B 0,C 180,E1 25684.081,E2 25684.081} C_VEL
LIN {X 0,Y 688.521,Z 1066.5,A -85,B 0,C 180,E1 25682.898,E2 25682.898} C_VEL
LIN {X 0,Y 687.063,Z 1091.27,A -85,B 0,C 180,E1 25681.303,E2 25681.303} C_VEL
LIN {X 0,Y 685.983,Z 1110.464,A -85,B 0,C 180,E1 25679.902,E2 25679.902} C_VEL
LIN {X 0,Y 684.981,Z 1128.832,A -85,B 0,C 180,E1 25678.417,E2 25678.417} C_VEL
LIN {X 0,Y 683.8,Z 1150.124,A -85,B 0,C 180,E1 25676.488,E2 25676.488} C_VEL
LIN {X 0,Y 682.982,Z 1166.579,A -85,B 0,C 180,E1 25674.812,E2 25674.812} C_VEL
LIN {X 0,Y 682.199,Z 1183.093,A -85,B 0,C 180,E1 25672.948,E2 25672.948} C_VEL
LIN {X 0,Y 681.502,Z 1199.566,A -85,B 0,C 180,E1 25670.836,E2 25670.836} C_VEL
LIN {X 0,Y 681.048,Z 1212.259,A -85,B 0,C 180,E1 25669.003,E2 25669.003} C_VEL
LIN {X 0,Y 680.671,Z 1224.076,A -85,B 0,C 180,E1 25667.087,E2 25667.087} C_VEL
LIN {X 0,Y 680.348,Z 1236.618,A -85,B 0,C 180,E1 25664.731,E2 25664.731} C_VEL
LIN {X 0,Y 680.162,Z 1245.599,A -85,B 0,C 180,E1 25662.741,E2 25662.741} C_VEL
LIN {X 0,Y 680.028,Z 1252.576,A -85,B 0,C 180,E1 25660.936,E2 25660.936} C_VEL
LIN {X 0,Y 679.931,Z 1258.166,A -85,B 0,C 180,E1 25659.226,E2 25659.226} C_VEL
LIN {X 0,Y 679.922,Z 1263.259,A -85,B 0,C 180,E1 25657.353,E2 25657.353} C_VEL
LIN {X 0,Y 679.918,Z 1267.847,A -85,B 0,C 180,E1 25655.064,E2 25655.064} C_VEL
LIN {X 0,Y 679.913,Z 1270.571,A -85,B 0,C 180,E1 25652.868,E2 25652.868} C_VEL
LIN {X 0,Y 679.88,Z 1271.725,A -85,B 0,C 180,E1 25651.014,E2 25651.014} C_VEL
LIN {X 0,Y 679.863,Z 1271.817,A -85,B 0,C 180,E1 25649.244,E2 25649.244} C_VEL
LIN {X 0,Y 679.903,Z 1270.917,A -85,B 0,C 180,E1 25647.474,E2 25647.474} C_VEL
LIN {X 0,Y 679.912,Z 1268.87,A -85,B 0,C 180,E1 25645.532,E2 25645.532} C_VEL
LIN {X 0,Y 679.925,Z 1264.832,A -85,B 0,C 180,E1 25643.246,E2 25643.246} C_VEL
LIN {X 0,Y 679.939,Z 1259.219,A -85,B 0,C 180,E1 25641.035,E2 25641.035} C_VEL
LIN {X 0,Y 680.015,Z 1253.221,A -85,B 0,C 180,E1 25639.155,E2 25639.155} C_VEL
LIN {X 0,Y 680.145,Z 1246.35,A -85,B 0,C 180,E1 25637.35,E2 25637.35} C_VEL
LIN {X 0,Y 680.307,Z 1238.297,A -85,B 0,C 180,E1 25635.534,E2 25635.534} C_VEL
LIN {X 0,Y 680.536,Z 1228.066,A -85,B 0,C 180,E1 25633.53,E2 25633.53} C_VEL
LIN {X 0,Y 680.994,Z 1213.907,A -85,B 0,C 180,E1 25631.158,E2 25631.158} C_VEL
LIN {X 0,Y 681.43,Z 1201.161,A -85,B 0,C 180,E1 25629.294,E2 25629.294} C_VEL
LIN {X 0,Y 682.032,Z 1186.8,A -85,B 0,C 180,E1 25627.416,E2 25627.416} C_VEL
LIN {X 0,Y 682.882,Z 1168.836,A -85,B 0,C 180,E1 25625.34,E2 25625.34} C_VEL
LIN {X 0,Y 683.693,Z 1152.251,A -85,B 0,C 180,E1 25623.631,E2 25623.631} C_VEL
LIN {X 0,Y 684.776,Z 1132.855,A -85,B 0,C 180,E1 25621.83,E2 25621.83} C_VEL
LIN {X 0,Y 685.876,Z 1112.432,A -85,B 0,C 180,E1 25620.159,E2 25620.159} C_VEL
LIN {X 0,Y 686.933,Z 1093.916,A -85,B 0,C 180,E1 25618.794,E2 25618.794} C_VEL
LIN {X 0,Y 688.193,Z 1071.928,A -85,B 0,C 180,E1 25617.337,E2 25617.337} C_VEL
LIN {X 0,Y 689.536,Z 1048.197,A -85,B 0,C 180,E1 25615.967,E2 25615.967} C_VEL
LIN {X 0,Y 690.648,Z 1027.677,A -85,B 0,C 180,E1 25614.922,E2 25614.922} C_VEL
LIN {X 0,Y 691.674,Z 1007.684,A -85,B 0,C 180,E1 25614.02,E2 25614.02} C_VEL
LIN {X 0,Y 692.658,Z 986.973,A -85,B 0,C 180,E1 25613.201,E2 25613.201} C_VEL
LIN {X 0,Y 693.766,Z 961.433,A -85,B 0,C 180,E1 25612.337,E2 25612.337} C_VEL
LIN {X 0,Y 694.721,Z 934.167,A -85,B 0,C 180,E1 25611.603,E2 25611.603} C_VEL
LIN {X 0,Y 695.457,Z 909.604,A -85,B 0,C 180,E1 25611.091,E2 25611.091} C_VEL
LIN {X 0,Y 696.054,Z 881.805,A -85,B 0,C 180,E1 25610.67,E2 25610.67} C_VEL
LIN {X 0,Y 698.375,Z 657.242,A -85,B 0,C 180,E1 25607.845,E2 25607.845} C_VEL
LIN {X 0,Y 700.685,Z 451.537,A -85,B 0,C 180,E1 25605.174,E2 25605.174} C_VEL
LIN {X 0,Y 700.673,Z 440.298,A -85,B 0,C 180,E1 25605.014,E2 25605.014} C_VEL
LIN {X 0,Y 688.357,Z 422.165,A -85,B 0,C 180,E1 25603.715,E2 25603.715} C_VEL
LIN {X 0,Y 685.273,Z 417.526,A -85,B 0,C 180,E1 25603.355,E2 25603.355} C_VEL
LIN {X 0,Y 682.201,Z 410.447,A -85,B 0,C 180,E1 25602.507,E2 25602.507} C_VEL
LIN {X 0,Y 680.552,Z 406.919,A -85,B 0,C 180,E1 25602.065,E2 25602.065} C_VEL
LIN {X 0,Y 680.472,Z 406.451,A -85,B 0,C 180,E1 25601.975,E2 25601.975} C_VEL
LIN {X 0,Y 680.464,Z 406.47,A -85,B 0,C 180,E1 25599.296,E2 25599.296} C_VEL
LIN {X 0,Y 680.527,Z 406.463,A -85,B 0,C 180,E1 25596.308,E2 25596.308} C_VEL
LIN {X 0,Y 680.456,Z 406.457,A -85,B 0,C 180,E1 25593.43,E2 25593.43} C_VEL
LIN {X 0,Y 680.479,Z 406.454,A -85,B 0,C 180,E1 25590.738,E2 25590.738} C_VEL
LIN {X 0,Y 680.477,Z 406.462,A -85,B 0,C 180,E1 25587.572,E2 25587.572} C_VEL
LIN {X 0,Y 680.451,Z 406.447,A -85,B 0,C 180,E1 25584.944,E2 25584.944} C_VEL
LIN {X 0,Y 680.524,Z 406.459,A -85,B 0,C 180,E1 25582.095,E2 25582.095} C_VEL
